(* CODESYS project tc3_harman_mesv2.6.10.library
   Author: Biro Csaba Attila
   Placeholder: Tc3_Harman_MES_Interface
   Title: Tc3_Harman_MES_Interface
   Version: 2.6.10
   Description: SAP-ME MES system interface library.
   Company: Harman

Project tree, tasks and I/O mapping:
  libraries: Tc2_Standard, * (Beckhoff Automation GmbH); Tc2_System, * (Beckhoff Automation GmbH); Tc2_TcpIp, * (Beckhoff Automation GmbH); Tc2_Utilities, * (Beckhoff Automation GmbH); Tc3_JsonXml, * (Beckhoff Automation GmbH); Tc3_Module, * (Beckhoff Automation GmbH); Tc3_Utilities_Extension, * (Harman)
  DUTs/
    data type E_TEST_STATE
    data type ENUM_MES_STATE
    data type ST_ASSEMBLY
    data type ST_ASSY_INFO
    data type ST_BOM
    data type ST_BOM_COMPONENT
    data type ST_GET_OP_STATE
    data type ST_INVENTORY
    data type ST_INVENTORY_LIST
    data type ST_MATERIAL
    data type ST_MATERIAL_INFO
    data type ST_MESDAT
    data type ST_MESDAT_ELEMENT
    data type ST_REQUEST
    data type ST_SET_ASSEMBLY
    data type ST_SHOPORDER
    data type ST_SHOPORDER_LIST
  FBs/
    function block FB_MES_INTERFACE_V2 [ST]: EXIT_SERVICE, GET_SERVICE_CONFIG, HIDE_SERVICE, LOCAL_INIT_SERVICE, REMOTE_INIT_SERVICE, SHOW_SERVICE, ASSY_ADD_MESDAT, ASSY_SAVE_MESDAT, ASSY_ADD_NCDAT, ASSY_SAVE_NCDAT, ASSEMBLE_BY_INVENTORY_LIST, CHECK_TIME_CONTROL, COMPLETE_SFC, GENERATE_SFC_BY_SO_AND_START, GET_CURRENT_OPERATION_STATE, GET_CUSTOM_DATA_BY_KEY, GET_INVENTORY_PARENT, GET_MAT_CUSTOM_DATA, GET_RECIPE_NAME_BY_OPERATION_JSON, GET_RECIPE_NAME_BY_OPERATION_XML, GET_SHOPORDER_BY_MAT, GET_TOTAL_BOM_BY_SO, IMPORT_AND_START_SFC, IMPORT_SFC, IS_VALID_INVENTORY_AND_IMPORT, MTERIAL_SETUP, SAVE_SFC_DATA, SCRAP_SFC, SIGNOFF_SFC, START_SFC, STOP_TIME_CONTROL, VALIDATE_IN_BOM, CREATE_XML_METH, GET_LOCAL_TIME, READ_XML_METH, FB_CALL_ACT
  FCs/
    function FC_GET_MATERIAL_FROM_HANDLE [ST]
    function FC_GET_REVISION_FROM_HANDLE [ST]
    function FC_REMOVE_HEADER [ST]
    function FC_REMOVE_STRING [ST]
  GVLs/
    global variables CONST_GVL
  TESTs/
    function GENERATE_MESDAT [ST]
    function GENERATE_NCDAT [ST]
    program HCP3_TEST_POU [ST]: FB_CALL_ACT
    program TEST_POU_1026_REPAIR [ST]: FB_CALL_ACT
    program TEST_POU_3026_SAVE_CF [ST]: FB_CALL_ACT
*)

// DUTs/E_TEST_STATE
TYPE E_TEST_STATE :
(
	PASSED:= 0,
	FAILED:= 1
):=FAILED;
END_TYPE

// DUTs/ENUM_MES_STATE
TYPE ENUM_MES_STATE :
(
	E_IDLE,
	E_CONNECTING,
	E_REQUEST_PROCESSING,
	E_REQUEST_PROCESSED,
	E_REQUEST_SEND,
	E_RESPONSE_RECIVED,
	E_RESPONSE_PROCESSING,
	E_RESPONSE_PROCESSED,
	E_DISCONNECTING,
	E_DONE,	
	E_ERROR		
):=E_IDLE;
END_TYPE

// DUTs/ST_ASSEMBLY
TYPE ST_ASSEMBLY :
STRUCT
	ASSEMBLY_READY		:STRING;
	ASSEMBLY_DONE		:STRING;
END_STRUCT
END_TYPE

// DUTs/ST_ASSY_INFO
TYPE ST_ASSY_INFO :
STRUCT
	ELEMENT:			ARRAY[1..9] OF ST_SET_ASSEMBLY;
END_STRUCT
END_TYPE

// DUTs/ST_BOM
TYPE ST_BOM :
STRUCT
	BOM_HANDLE:					STRING;
	BOMSTATUS:					STRING;
	DESCRIPTION:				STRING;
	SHOPORDER:					STRING;
	BOM_COMPONENTS:				ARRAY[0..19] OF ST_BOM_COMPONENT;
END_STRUCT
END_TYPE

// DUTs/ST_BOM_COMPONENT
TYPE ST_BOM_COMPONENT :
STRUCT
	BOM_COMPONENT_TYPE:				STRING;
	MATERIALS:						ARRAY[0..9] OF ST_MATERIAL;
	OPERATION:						STRING;
	QUANTITY:						STRING;
	SEQUENCE: 						STRING;
END_STRUCT
END_TYPE

// DUTs/ST_GET_OP_STATE
TYPE ST_GET_OP_STATE :
STRUCT
	ARCHIVE:		STRING;
	OP_INDEX:		STRING;
	OP_NAME:		STRING;
	SFC_STATE:		STRING;	
	OPEN_NC:		STRING;
	MAT_NO:			STRING;	
	REVISION:		STRING;
END_STRUCT
END_TYPE

// DUTs/ST_INVENTORY
TYPE ST_INVENTORY :
STRUCT
	DONE:			STRING;
	MAT_NO:			STRING;	
	REVISION:		STRING;
	SFC:			STRING;
	VALUES:			STRING;
END_STRUCT
END_TYPE

// DUTs/ST_INVENTORY_LIST
TYPE ST_INVENTORY_LIST :
STRUCT
	LIST:		ARRAY[0..9] OF ST_INVENTORY;
END_STRUCT
END_TYPE

// DUTs/ST_MATERIAL
TYPE ST_MATERIAL :
STRUCT
	MATERIAL:			STRING;
	REVISION:			STRING;
END_STRUCT
END_TYPE

// DUTs/ST_MATERIAL_INFO
TYPE ST_MATERIAL_INFO :
STRUCT
	MATNO:					STRING;
	REVISION:				STRING;
	SHOPORDER:				STRING;
	OPERATION:				STRING;
	RELEASECOUNT:			STRING;
END_STRUCT
END_TYPE

// DUTs/ST_MESDAT
TYPE ST_MESDAT :
STRUCT
	N:			INT;
	MESDAT:		ARRAY[1..200] OF ST_MESDAT_ELEMENT;
END_STRUCT
END_TYPE

// DUTs/ST_MESDAT_ELEMENT
TYPE ST_MESDAT_ELEMENT :
STRUCT
	RESPONSE_CODE:			STRING;		(* required in NC Data log - Error Id *)
	RESPONSE_DESCRIPTION:	STRING;		(* optional - Error description in NC Data log equal with DESCR *)
	CLIENT_DATE:			STRING;		(* required - Use the GET_LOCAL_TIME() method for generate in proper format. *)
	TEST_STATE:				STRING;		(* required - Use E_TEST_STATE value as string. *)
	TEST_STEP:				STRING;		(* required - Id of test step, (screw no, camera step...) *)
	DESCR:					STRING;		(* optional - Process step description, Error description in NC Data log *)
	UNIT:					STRING;		(* optional - Measurement unit *)
	VALUE:					STRING;		(* required - Measured data, if it Pass/Fail data only use 0 or 1 *)
	LL:						STRING;		(* optional - Lower limit *)
	UL:						STRING;		(* optional - Upper limit *)
END_STRUCT
END_TYPE

// DUTs/ST_REQUEST
TYPE ST_REQUEST :
STRUCT
	RESP_ACTION:		STRING;
	RESP_CODE:			STRING;
	ERR_MSG:			STRING[255];
END_STRUCT
END_TYPE

// DUTs/ST_SET_ASSEMBLY
TYPE ST_SET_ASSEMBLY :
STRUCT
	SFC:				STRING;
	MATNO:				STRING;
	REVISION:			STRING;
	INVENTORYID:		STRING;
	OPERATION:			STRING;
	RESOURCE:			STRING;
	DESCRIPTION:		STRING;
	BOM:				STRING;
	BOMREV:				STRING;
	SEQUENCE:			STRING;
	DATEASSEMBLED:		STRING;
	STRUCTUREPOSITION:	STRING;
	
	(*
	       <SET-ASSEMBLY>
            <SFC>614790420198010103089851</SFC>
            <MATNO>00003089851</MATNO>
            <REVISION>001</REVISION>
            <INVENTORYID>614790420198010103089851</INVENTORYID>
            <OPERATION>OP_ASSEMBLY_1</OPERATION>
            <RESOURCE>R_HUSZP5BRAFA11</RESOURCE>
            <DESCRIPTION>HOUSING HIGH RAM  B279 C1</DESCRIPTION>
            <BOM>00003561631_056</BOM>
            <BOMREV>001</BOMREV>
            <SEQUENCE>10</SEQUENCE>
            <DATEASSEMBLED>2/10/2020 10:59:04 PM</DATEASSEMBLED>
            <STRUCTUREPOSITION>0.0</STRUCTUREPOSITION>
          </SET-ASSEMBLY>
	*)
END_STRUCT
END_TYPE

// DUTs/ST_SHOPORDER
TYPE ST_SHOPORDER :
STRUCT
	HANDLE:				STRING;
	RELEASED:			STRING;
	STATUS:				STRING;
	QUANTITY:			STRING;
	SHOPORDER_TYPE:		STRING;
END_STRUCT
END_TYPE

// DUTs/ST_SHOPORDER_LIST
TYPE ST_SHOPORDER_LIST :
STRUCT
	LIST:		ARRAY[0..9] OF ST_SHOPORDER;
END_STRUCT
END_TYPE

// GVLs/CONST_GVL
VAR_GLOBAL CONSTANT
	DEFAULT_PRG_NAME:			STRING:='TwinCat3 - Build:v4024.17';
	DEFAULT_PRG_REV:			STRING:='v2.6.9';
END_VAR

// FBs/FB_MES_INTERFACE_V2
FUNCTION_BLOCK FB_MES_INTERFACE_V2
VAR_INPUT
	HOST:				T_IPV4ADDR := '';
	PORT:				UDINT;
	ENABLE:				BOOL;
	RESET:				BOOL;
	STX:				BYTE:= TCP_GVL.DEFAULT_STX;
	ETX:				BYTE:= TCP_GVL.DEFAULT_ETX;
	RESP:				REFERENCE TO ST_REQUEST;
	
	TEST_ADAPTER:		STRING;		//Adapter ID (Code)
	ADAPTER_ID:			STRING;		//Nest no. (1-5)
END_VAR
VAR_OUTPUT
	BUSY:				BOOL;
	READY:				BOOL;
	DONE:				BOOL;
	INTERFACE_CLOSED:	BOOL:=TRUE;
	ERROR:				BOOL;
	ERROR_ID:			UDINT;
END_VAR
VAR
	FB_TCP_IP_CLIENT:				FB_TCP_IP_CLIENT_LDAT;
	STATE:							ENUM_MES_STATE;
	
	INTERFACE_DIR:					STRING:='C:\Program Files\Harman\SAP-ME Interface';
	INTERFACE_FILE:					STRING:='SAP-ME Interface.exe';
	INTERFACE_ARG:					STRING:='initHMIAssy';
	
	EXECUTE:						BOOL;
	LOCAL_INIT:						BOOL;
	INIT:							BOOL;
	CB_MESSAGE:						UDINT;
	RT_EXECUTE, RT_RESET, RT_TCP_ERROR:R_TRIG;
	SYS_TIME_FB:					FB_LocalSystemTime;
	REQUEST_STRING:					STRING[DEFAULT_LDAT_LENGTH]:='';			
	RESPONSE_STRING:				STRING[DEFAULT_LDAT_LENGTH]:='';
	
	//================ XML =================
	FB_XML_PARSER: 			FB_XmlDomParser;
	OBJ_ROOT: 				SXmlNode;		
	
	// Base XML tags
	XML_HMIXML: 			SXmlNode;
	XML_PACKET: 			SXmlNode;	
	XML_BASICS: 			SXmlNode;		
	XML_ACTION: 			SXmlNode;
	XML_ARGUMENTS: 			SXmlNode;
	XML_RESULTS: 			SXmlNode;	
	XML_MSG: 				SXmlNode;	
	
	// Base response XML tags
	XML_RESCODE: 			SXmlNode;	
	XML_RESSTANDARDMESSAGE: SXmlNode;
	
	// Temporary container of RESTINFO for a later querys	
	XML_RESTINFO:			SXmlNode;
	
	// Request result inforamtion ErrorMessage, ResponseCode...
	XML_REQUEST_RESULT:		ST_REQUEST;	
	DEBUG:					STRING(10000);
	
	TP_RECONNECT:			TP;
	TON_INIT:				TON;
	FB_START_INTERFACE:		NT_StartProcess;
	eSubSystem: 			E_SubSystem:= E_SubSystem.LOGIC;
	FB_LOGGER:				FB_EventLogger:= (eSubsystem:= eSubsystem);
END_VAR

RT_EXECUTE(CLK:=EXECUTE);
RT_RESET(CLK:=RESET);
TP_RECONNECT(IN:=(FB_TCP_IP_CLIENT.CONNECTION_STATE<>ESOCKET_CONNECTED OR FB_TCP_IP_CLIENT.ERROR), PT:=T#250MS);
TON_INIT(IN:=INIT);	(* Delay for get configuration call *)
SYS_TIME_FB(bEnable:=TRUE,dwCycle:=1);

IF FB_TCP_IP_CLIENT.ERROR_ID<>0 THEN
	ERROR_ID:=FB_TCP_IP_CLIENT.ERROR_ID;
END_IF

BUSY:= STATE<>E_IDLE OR LOCAL_INIT OR INIT;
READY:= STATE=E_IDLE AND NOT INIT AND NOT INTERFACE_CLOSED;
ERROR:= STATE=E_ERROR;

IF RT_RESET.Q THEN
	//FB_LOGGER(sMsg:=CONCAT('Reseted externaly - ERROR_ID: ', UDINT_TO_STRING(ERROR_ID)), eSevr:=TcEventSeverity.Info);
	EXECUTE:=FALSE;
	ERROR_ID:= 0;
	STATE:=E_IDLE;
	REQUEST_STRING:= '';
	RESPONSE_STRING:= '';
	RESP.ERR_MSG:='';
	RESP.RESP_ACTION:='';
	RESP.RESP_CODE:='';
END_IF

(* Get MES configuration from interface *)
IF INIT THEN
	IF GET_SERVICE_CONFIG() THEN
		LOCAL_INIT:=FALSE;
		INIT:=FALSE;
	END_IF
END_IF

CASE STATE OF
	E_IDLE:
		IF RT_EXECUTE.Q THEN
			FB_TCP_IP_CLIENT.ENABLE:=TRUE;
			DONE:=FALSE;
			REQUEST_STRING:='';
			RESPONSE_STRING:='';
			CREATE_XML_METH();
			STATE:=E_CONNECTING;
		END_IF	
	E_CONNECTING:
		IF FB_TCP_IP_CLIENT.CONNECTION_STATE=ESOCKET_CONNECTED AND FB_TCP_IP_CLIENT.READY AND NOT FB_TCP_IP_CLIENT.BUSY THEN
			STATE:=E_REQUEST_PROCESSING;
		END_IF
		
	E_REQUEST_SEND:
		CB_MESSAGE:= FB_XML_PARSER.CopyDocument(REQUEST_STRING, SIZEOF(REQUEST_STRING));
		IF FB_TCP_IP_CLIENT.SEND(REQUEST_STRING, CB_MESSAGE, RESPONSE_STRING) THEN
			STATE:= E_RESPONSE_RECIVED;
		END_IF
		
	E_RESPONSE_RECIVED:
		READ_XML_METH();
		STATE:= E_RESPONSE_PROCESSING;
		MEMCPY(ADR(RESP),ADR(XML_REQUEST_RESULT), SIZEOF(XML_REQUEST_RESULT));
		
	E_DISCONNECTING:
		FB_TCP_IP_CLIENT.ENABLE:=FALSE;
		IF FB_TCP_IP_CLIENT.CONNECTION_STATE=ESOCKET_CONNECTED THEN
			STATE:=E_DONE;
		END_IF
	E_DONE:
		DONE:=TRUE;
		IF NOT EXECUTE THEN
			STATE:= E_IDLE;
		END_IF
		
	E_ERROR:
		//FB_LOGGER(sMsg:=CONCAT(CONCAT(CONCAT(CONCAT(CONCAT('Process done with issue. ERROR_ID: ', UDINT_TO_STRING(ERROR_ID)), ' Error message: '), XML_REQUEST_RESULT.ERR_MSG), ' Response code: '), XML_REQUEST_RESULT.RESP_CODE), eSevr:=TcEventSeverity.Error);
		EXECUTE:=FALSE;
		DONE:=FALSE;
		
END_CASE

IF ERROR_ID <> 0 THEN
	STATE:= E_ERROR;
END_IF

FB_CALL_ACT();

METHOD PUBLIC EXIT_SERVICE : BOOL
VAR
	XML_NODE:			SXmlNode;
END_VAR
CASE STATE OF
	E_IDLE:
		EXECUTE:=TRUE;
		
	E_REQUEST_PROCESSING:
		DEBUG:='';
		FB_XML_PARSER.AppendAttributeAsInt(XML_HMIXML,'operationIndex',0);
		FB_XML_PARSER.AppendAttributeAsInt(XML_HMIXML,'serviceId',2);		
		FB_XML_PARSER.SetChild(XML_ACTION,'1000001',FALSE);
		FB_XML_PARSER.CopyDocument(REQUEST_STRING, SIZEOF(REQUEST_STRING));
		STATE:= E_REQUEST_SEND;
		
	E_RESPONSE_PROCESSING:
		IF XML_REQUEST_RESULT.RESP_CODE = '0' THEN
			XML_RESTINFO:=FB_XML_PARSER.ChildByName(XML_RESULTS, 'RESTINFO');
			EXECUTE:=FALSE;
			STATE:= E_DISCONNECTING;
		ELSE
			MEMCPY(ADR(RESP),ADR(XML_REQUEST_RESULT), SIZEOF(XML_REQUEST_RESULT));
			ADSLOGSTR(ADSLOG_MSGTYPE_ERROR OR ADSLOG_MSGTYPE_LOG, 'SAP-ME error occured RESCODE: %s', CONCAT(CONCAT(RESP.RESP_CODE, ' ERR_MSG: '), RESP.ERR_MSG));
			EXECUTE:=FALSE;
			STATE:= E_DISCONNECTING;
		END_IF
	E_DONE: INTERFACE_CLOSED:=TRUE;
END_CASE
EXIT_SERVICE:= (STATE=E_DONE);
END_METHOD

METHOD PUBLIC GET_SERVICE_CONFIG : BOOL
VAR
	XML_NODE:			SXmlNode;
END_VAR
CASE STATE OF
	E_IDLE:
		EXECUTE:=TRUE;
		
	E_REQUEST_PROCESSING:
		DEBUG:='';
		FB_XML_PARSER.AppendAttributeAsInt(XML_HMIXML,'operationIndex',0);
		FB_XML_PARSER.AppendAttributeAsInt(XML_HMIXML,'serviceId',2);		
		FB_XML_PARSER.SetChild(XML_ACTION,'1000000',FALSE);
		FB_XML_PARSER.CopyDocument(REQUEST_STRING, SIZEOF(REQUEST_STRING));
		STATE:= E_REQUEST_SEND;
		
	E_RESPONSE_PROCESSING:
		IF XML_REQUEST_RESULT.RESP_CODE = '0' THEN
			XML_RESTINFO:=FB_XML_PARSER.ChildByName(XML_RESULTS, 'RESTINFO');
			EXECUTE:=FALSE;
			STATE:= E_DISCONNECTING;
		ELSE
			MEMCPY(ADR(RESP),ADR(XML_REQUEST_RESULT), SIZEOF(XML_REQUEST_RESULT));
			ADSLOGSTR(ADSLOG_MSGTYPE_ERROR OR ADSLOG_MSGTYPE_LOG, 'SAP-ME error occured RESCODE: %s', CONCAT(CONCAT(RESP.RESP_CODE, ' ERR_MSG: '), RESP.ERR_MSG));
			EXECUTE:=FALSE;
			STATE:= E_DISCONNECTING;
		END_IF
END_CASE
GET_SERVICE_CONFIG:= (STATE=E_DONE);
END_METHOD

METHOD PUBLIC HIDE_SERVICE : BOOL
VAR
	XML_NODE:			SXmlNode;
END_VAR
CASE STATE OF
	E_IDLE:
		EXECUTE:=TRUE;
		
	E_REQUEST_PROCESSING:
		DEBUG:='';
		FB_XML_PARSER.AppendAttributeAsInt(XML_HMIXML,'operationIndex',0);
		FB_XML_PARSER.AppendAttributeAsInt(XML_HMIXML,'serviceId',2);		
		FB_XML_PARSER.SetChild(XML_ACTION,'1000003',FALSE);
		FB_XML_PARSER.CopyDocument(REQUEST_STRING, SIZEOF(REQUEST_STRING));
		STATE:= E_REQUEST_SEND;
		
	E_RESPONSE_PROCESSING:
		IF XML_REQUEST_RESULT.RESP_CODE = '0' THEN
			XML_RESTINFO:=FB_XML_PARSER.ChildByName(XML_RESULTS, 'RESTINFO');
			EXECUTE:=FALSE;
			STATE:= E_DISCONNECTING;
		ELSE
			MEMCPY(ADR(RESP),ADR(XML_REQUEST_RESULT), SIZEOF(XML_REQUEST_RESULT));
			ADSLOGSTR(ADSLOG_MSGTYPE_ERROR OR ADSLOG_MSGTYPE_LOG, 'SAP-ME error occured RESCODE: %s', CONCAT(CONCAT(RESP.RESP_CODE, ' ERR_MSG: '), RESP.ERR_MSG));
			EXECUTE:=FALSE;
			STATE:= E_DISCONNECTING;
		END_IF
	E_DONE: INTERFACE_CLOSED:=TRUE;
END_CASE
HIDE_SERVICE:= (STATE=E_DONE);
END_METHOD

METHOD PUBLIC LOCAL_INIT_SERVICE : BOOL
LOCAL_INIT:=TRUE;
TON_INIT.PT:=T#3S;
INIT:=TRUE;
INTERFACE_CLOSED:=FALSE;
LOCAL_INIT_SERVICE:= STATE=E_DONE;
END_METHOD

METHOD PUBLIC REMOTE_INIT_SERVICE : BOOL
INIT:=TRUE;
TON_INIT.PT:=T#0S;
INTERFACE_CLOSED:=FALSE;
REMOTE_INIT_SERVICE:= STATE=E_DONE;
END_METHOD

METHOD PUBLIC SHOW_SERVICE : BOOL
VAR
	XML_NODE:			SXmlNode;
END_VAR
CASE STATE OF
	E_IDLE:
		EXECUTE:=TRUE;
		
	E_REQUEST_PROCESSING:
		DEBUG:='';
		FB_XML_PARSER.AppendAttributeAsInt(XML_HMIXML,'operationIndex',0);
		FB_XML_PARSER.AppendAttributeAsInt(XML_HMIXML,'serviceId',2);		
		FB_XML_PARSER.SetChild(XML_ACTION,'1000002',FALSE);
		FB_XML_PARSER.CopyDocument(REQUEST_STRING, SIZEOF(REQUEST_STRING));
		STATE:= E_REQUEST_SEND;
		
	E_RESPONSE_PROCESSING:
		IF XML_REQUEST_RESULT.RESP_CODE = '0' THEN
			XML_RESTINFO:=FB_XML_PARSER.ChildByName(XML_RESULTS, 'RESTINFO');
			EXECUTE:=FALSE;
			STATE:= E_DISCONNECTING;
		ELSE
			MEMCPY(ADR(RESP),ADR(XML_REQUEST_RESULT), SIZEOF(XML_REQUEST_RESULT));
			ADSLOGSTR(ADSLOG_MSGTYPE_ERROR OR ADSLOG_MSGTYPE_LOG, 'SAP-ME error occured RESCODE: %s', CONCAT(CONCAT(RESP.RESP_CODE, ' ERR_MSG: '), RESP.ERR_MSG));
			EXECUTE:=FALSE;
			STATE:= E_DISCONNECTING;
		END_IF
	E_DONE: INTERFACE_CLOSED:=TRUE;
END_CASE
SHOW_SERVICE:= (STATE=E_DONE);
END_METHOD

METHOD PUBLIC ASSY_ADD_MESDAT : BOOL
VAR_INPUT
	DATA:				REFERENCE TO ST_MESDAT_ELEMENT;
END_VAR
VAR
	XML_SET:			SXmlNode;
	XML_CLIENTDATE:		SXmlNode;
	XML_TESTSTATE:		SXmlNode;
	XML_TESTSTEP:		SXmlNode;	
	XML_DESCR:			SXmlNode;
	XML_TESTVALUE:		SXmlNode;		
	XML_UNIT:			SXmlNode;	
	XML_LOWERLIMIT:		SXmlNode;	
	XML_UPPERLIMIT:		SXmlNode;	
END_VAR
ASSY_ADD_MESDAT:=FALSE;
XML_SET := FB_XML_PARSER.AppendNode(XML_ARGUMENTS, 'SET');	
		
XML_CLIENTDATE := FB_XML_PARSER.AppendNode(XML_SET, 'CLIENTDATE'); //Req
XML_TESTSTATE := FB_XML_PARSER.AppendNode(XML_SET, 'TESTSTATE');//Req
XML_TESTSTEP := FB_XML_PARSER.AppendNode(XML_SET, 'TESTSTEP');//Req
XML_DESCR := FB_XML_PARSER.AppendNode(XML_SET, 'DESCR'); //Optional
XML_TESTVALUE := FB_XML_PARSER.AppendNode(XML_SET, 'TESTVALUE');//Req
XML_UNIT := FB_XML_PARSER.AppendNode(XML_SET, 'UNIT');	//Optional
XML_LOWERLIMIT := FB_XML_PARSER.AppendNode(XML_SET, 'LOWERLIMIT'); //Optional
XML_UPPERLIMIT := FB_XML_PARSER.AppendNode(XML_SET, 'UPPERLIMIT'); //Optional

FB_XML_PARSER.SetChild(XML_CLIENTDATE, DATA.CLIENT_DATE, FALSE);
FB_XML_PARSER.SetChild(XML_TESTSTATE,DATA.TEST_STATE, FALSE);			
FB_XML_PARSER.SetChild(XML_TESTSTEP, DATA.TEST_STEP, FALSE);					
FB_XML_PARSER.SetChild(XML_DESCR, DATA.DESCR, FALSE);				
FB_XML_PARSER.SetChild(XML_TESTVALUE, DATA.VALUE, FALSE);					
FB_XML_PARSER.SetChild(XML_UNIT, DATA.UNIT, FALSE);							
FB_XML_PARSER.SetChild(XML_LOWERLIMIT, DATA.LL, FALSE);							
FB_XML_PARSER.SetChild(XML_UPPERLIMIT, DATA.UL, FALSE);

ASSY_ADD_MESDAT:=TRUE;
END_METHOD

METHOD PUBLIC ASSY_SAVE_MESDAT : BOOL
VAR_INPUT
	SFC:					STRING;					//Product Serial Number
	INDEX:					INT;					//Operation index
	DATA:					REFERENCE TO ST_MESDAT;	//Measurement data.	
END_VAR
VAR_OUTPUT
	
END_VAR
VAR
	XML_NODE:				SXmlNode;
	XML_TESTADAPTER:		SXmlNode;
	XML_ADAPTERID:			SXmlNode;
	XML_PROGRAMNAME: 		SXmlNode;	
	XML_PROGREV:			SXmlNode;
			
	CNT:					INT:=1;
END_VAR
CASE STATE OF
	E_IDLE:
		IF DATA.N>=1 AND DATA.N<=200 THEN
			EXECUTE:=TRUE;
		ELSE
			// TODO: If data array is empty return and log error message.
			ASSY_SAVE_MESDAT:=TRUE;
		END_IF
		
	E_REQUEST_PROCESSING:		
		FB_XML_PARSER.AppendAttributeAsInt(XML_HMIXML,'operationIndex',INDEX);
		FB_XML_PARSER.AppendAttributeAsInt(XML_HMIXML,'serviceId',2);	
			
		XML_NODE:= FB_XML_PARSER.AppendNode(XML_ARGUMENTS, 'SFC');
		XML_TESTADAPTER:= FB_XML_PARSER.AppendNode(XML_ARGUMENTS, 'TESTADAPTER'); //Req
		XML_ADAPTERID:= FB_XML_PARSER.AppendNode(XML_ARGUMENTS, 'FIXTUREID'); //Req
		XML_PROGRAMNAME:= FB_XML_PARSER.AppendNode(XML_ARGUMENTS, 'PROGRAMID'); //Optional
		XML_PROGREV:= FB_XML_PARSER.AppendNode(XML_ARGUMENTS, 'PROGRAMREV'); //Optional
		
		FB_XML_PARSER.SetChild(XML_ACTION,'3523', FALSE);
		
		FB_XML_PARSER.SetChild(XML_NODE, SFC, FALSE);
		FB_XML_PARSER.SetChild(XML_TESTADAPTER, TEST_ADAPTER, FALSE);
		FB_XML_PARSER.SetChild(XML_ADAPTERID, ADAPTER_ID, FALSE);
		FB_XML_PARSER.SetChild(XML_PROGRAMNAME, DEFAULT_PRG_NAME, FALSE);	
		FB_XML_PARSER.SetChild(XML_PROGREV, DEFAULT_PRG_REV, FALSE);	
		
		FOR CNT:=1 TO (DATA.N) DO
			ASSY_ADD_MESDAT(DATA.MESDAT[CNT]);			
		END_FOR
		
		STATE:= E_REQUEST_SEND;
		
	E_RESPONSE_PROCESSING:
		IF XML_REQUEST_RESULT.RESP_CODE = '0' THEN		
			EXECUTE:=FALSE;
			STATE:= E_DISCONNECTING;
		ELSE
			MEMCPY(ADR(RESP),ADR(XML_REQUEST_RESULT), SIZEOF(XML_REQUEST_RESULT));
			ADSLOGSTR(ADSLOG_MSGTYPE_ERROR OR ADSLOG_MSGTYPE_LOG, 'SAP-ME error occured RESCODE: %s', CONCAT(CONCAT(RESP.RESP_CODE, ' ERR_MSG: '), RESP.ERR_MSG));
			EXECUTE:=FALSE;
			STATE:= E_DISCONNECTING;
		END_IF

END_CASE
ASSY_SAVE_MESDAT:= (STATE=E_DONE);
END_METHOD

METHOD PUBLIC ASSY_ADD_NCDAT : BOOL
VAR_INPUT
	DATA:				REFERENCE TO ST_MESDAT_ELEMENT;
END_VAR
VAR
	XML_SET:			SXmlNode;
	XML_TESTSTATE:		SXmlNode;
	XML_TESTSTEP:		SXmlNode;	
	XML_RESPCODE:		SXmlNode;
	XML_RESPDESC:		SXmlNode;	
	XML_DESCR:			SXmlNode;
	XML_TESTVALUE:		SXmlNode;
	XML_LOWERLIMIT:		SXmlNode;	
	XML_UPPERLIMIT:		SXmlNode;	
END_VAR
ASSY_ADD_NCDAT:=FALSE;
XML_SET := FB_XML_PARSER.AppendNode(XML_ARGUMENTS, 'SET');	
		
XML_TESTSTATE := FB_XML_PARSER.AppendNode(XML_SET, 'TESTSTATE');
XML_TESTSTEP := FB_XML_PARSER.AppendNode(XML_SET, 'TESTSTEP');
XML_RESPCODE := FB_XML_PARSER.AppendNode(XML_SET, 'RESPONSECODE');
XML_RESPDESC := FB_XML_PARSER.AppendNode(XML_SET, 'RESPONSECODEDESCR');
XML_DESCR := FB_XML_PARSER.AppendNode(XML_SET, 'DESCR');
XML_TESTVALUE := FB_XML_PARSER.AppendNode(XML_SET, 'TESTVALUE');
XML_LOWERLIMIT := FB_XML_PARSER.AppendNode(XML_SET, 'LOWERLIMIT');
XML_UPPERLIMIT := FB_XML_PARSER.AppendNode(XML_SET, 'UPPERLIMIT');

FB_XML_PARSER.SetChild(XML_TESTSTATE, DATA.TEST_STATE, FALSE);			
FB_XML_PARSER.SetChild(XML_TESTSTEP, DATA.TEST_STEP, FALSE);
FB_XML_PARSER.SetChild(XML_RESPCODE, DATA.RESPONSE_CODE, FALSE);			
FB_XML_PARSER.SetChild(XML_RESPDESC, DATA.RESPONSE_DESCRIPTION, FALSE);					
FB_XML_PARSER.SetChild(XML_DESCR, DATA.DESCR, FALSE);				
FB_XML_PARSER.SetChild(XML_TESTVALUE, DATA.VALUE, FALSE);					
FB_XML_PARSER.SetChild(XML_LOWERLIMIT, DATA.LL, FALSE);							
FB_XML_PARSER.SetChild(XML_UPPERLIMIT, DATA.UL, FALSE);	

ASSY_ADD_NCDAT:=TRUE;
END_METHOD

METHOD PUBLIC ASSY_SAVE_NCDAT : BOOL
VAR_INPUT
	SFC:					STRING;					//Product Serial Number
	INDEX:					INT;					//Operation index
	DATA:					REFERENCE TO ST_MESDAT;	//Measurement data.	
END_VAR
VAR_OUTPUT
	
END_VAR
VAR
	XML_SFC:				SXmlNode;
	XML_TESTADAPTER:		SXmlNode;
	XML_ADAPTERID:			SXmlNode;
	XML_CLIENTDATE:			SXmlNode;
	CLIENT_DATE:			STRING;	
	CNT:					INT:=1;
END_VAR
CLIENT_DATE:= GET_LOCAL_TIME();
CASE STATE OF
	E_IDLE:
		IF DATA.N>=1 AND DATA.N<=200 THEN
			EXECUTE:=TRUE;
		ELSE
			// TODO: If data array is empty generate unknown error... just for fail safe NC Logging
			DATA.N:=1;
			DATA.MESDAT[1].CLIENT_DATE:=GET_LOCAL_TIME();
			DATA.MESDAT[1].DESCR:='Unknown TwinCAT error - No data found in NC-Data container.';
			DATA.MESDAT[1].LL:='0';
			DATA.MESDAT[1].RESPONSE_CODE:='16003';
			DATA.MESDAT[1].RESPONSE_DESCRIPTION:='Unknown TwinCAT error - No data found in NC-Data container.';
			DATA.MESDAT[1].TEST_STATE:='1';
			DATA.MESDAT[1].TEST_STEP:='-1';
			DATA.MESDAT[1].UL:='0';
			DATA.MESDAT[1].UNIT:='Dig';
			DATA.MESDAT[1].VALUE:='-1';
			
			EXECUTE:=TRUE;
		END_IF
		
	E_REQUEST_PROCESSING:		
		CLIENT_DATE:=GET_LOCAL_TIME();
		FB_XML_PARSER.AppendAttributeAsInt(XML_HMIXML,'operationIndex',INDEX);
		FB_XML_PARSER.AppendAttributeAsInt(XML_HMIXML,'serviceId',2);	
			
		XML_SFC:= FB_XML_PARSER.AppendNode(XML_ARGUMENTS, 'SFC');
		XML_CLIENTDATE := FB_XML_PARSER.AppendNode(XML_ARGUMENTS, 'CLIENTDATE');
		XML_TESTADAPTER:= FB_XML_PARSER.AppendNode(XML_ARGUMENTS, 'TESTADAPTER');
		XML_ADAPTERID:= FB_XML_PARSER.AppendNode(XML_ARGUMENTS, 'FIXTUREID');
		
		FB_XML_PARSER.SetChild(XML_ACTION,'3503', FALSE);
		
		FB_XML_PARSER.SetChild(XML_SFC, SFC, FALSE);
		FB_XML_PARSER.SetChild(XML_CLIENTDATE, CLIENT_DATE, FALSE);
		FB_XML_PARSER.SetChild(XML_TESTADAPTER, TEST_ADAPTER, FALSE);
		FB_XML_PARSER.SetChild(XML_ADAPTERID, ADAPTER_ID, FALSE);	
		
		FOR CNT:=1 TO (DATA.N) DO
			ASSY_ADD_NCDAT(DATA.MESDAT[CNT]);			
		END_FOR
		
		STATE:= E_REQUEST_SEND;
		
	E_RESPONSE_PROCESSING:
		IF XML_REQUEST_RESULT.RESP_CODE = '0' THEN		
			EXECUTE:=FALSE;
			STATE:= E_DISCONNECTING;
		ELSE
			MEMCPY(ADR(RESP),ADR(XML_REQUEST_RESULT), SIZEOF(XML_REQUEST_RESULT));
			ADSLOGSTR(ADSLOG_MSGTYPE_ERROR OR ADSLOG_MSGTYPE_LOG, 'SAP-ME error occured RESCODE: %s', CONCAT(CONCAT(RESP.RESP_CODE, ' ERR_MSG: '), RESP.ERR_MSG));
			EXECUTE:=FALSE;
			STATE:= E_DISCONNECTING;
		END_IF

END_CASE
ASSY_SAVE_NCDAT:= (STATE=E_DONE);
END_METHOD

METHOD PUBLIC ASSEMBLE_BY_INVENTORY_LIST : BOOL
VAR_INPUT
	SFC:				STRING;
	INDEX:				INT;
	INVENTORY_LIST:		ST_INVENTORY_LIST;
END_VAR
VAR
	XML_NODE:			SXmlNode;
	XML_SET:			SXmlNode;
	XML_INVENTORY_ID:	SXmlNode;
	XML_INVENTORI_MAT:	SXmlNode;
	XML_INVENTORI_REV:	SXmlNode;
	
	CNT:				INT;
END_VAR
CASE STATE OF
	E_IDLE:
		EXECUTE:=TRUE;
		
	E_REQUEST_PROCESSING:
		DEBUG:='';
		FB_XML_PARSER.AppendAttributeAsInt(XML_HMIXML,'operationIndex',INDEX);
		FB_XML_PARSER.AppendAttributeAsInt(XML_HMIXML,'serviceId',2);		
		FB_XML_PARSER.SetChild(XML_ACTION,'2138',FALSE);
		XML_NODE := FB_XML_PARSER.AppendNode(XML_ARGUMENTS, 'SFC');
		FB_XML_PARSER.SetChild(XML_NODE,SFC,FALSE);
		FOR CNT:=0 TO 9 BY 1 DO
			IF INVENTORY_LIST.LIST[CNT].SFC<>'' AND LEN(INVENTORY_LIST.LIST[CNT].MAT_NO)=11 AND LEN(INVENTORY_LIST.LIST[CNT].REVISION)=3 THEN
				XML_SET := FB_XML_PARSER.AppendNode(XML_ARGUMENTS, 'SET');
					XML_INVENTORY_ID := FB_XML_PARSER.AppendNode(XML_SET, 'INVENTORYID');
					FB_XML_PARSER.SetChild(XML_INVENTORY_ID,INVENTORY_LIST.LIST[CNT].SFC,FALSE);
					XML_INVENTORI_MAT := FB_XML_PARSER.AppendNode(XML_SET, 'MATNO');
					FB_XML_PARSER.SetChild(XML_INVENTORI_MAT,INVENTORY_LIST.LIST[CNT].MAT_NO,FALSE);
					XML_INVENTORI_REV := FB_XML_PARSER.AppendNode(XML_SET, 'MATNO_REV');
					FB_XML_PARSER.SetChild(XML_INVENTORI_REV,INVENTORY_LIST.LIST[CNT].REVISION,FALSE);
			END_IF			
		END_FOR;
		
		FB_XML_PARSER.CopyDocument(REQUEST_STRING, SIZEOF(REQUEST_STRING));
		DEBUG:=REQUEST_STRING;
		STATE:= E_REQUEST_SEND;
		
	E_RESPONSE_PROCESSING:
		IF XML_REQUEST_RESULT.RESP_CODE = '0' THEN
			XML_RESTINFO:=FB_XML_PARSER.ChildByName(XML_RESULTS, 'RESTINFO');		
			EXECUTE:=FALSE;
			STATE:= E_DISCONNECTING;
		ELSE
			MEMCPY(ADR(RESP),ADR(XML_REQUEST_RESULT), SIZEOF(XML_REQUEST_RESULT));
			ADSLOGSTR(ADSLOG_MSGTYPE_ERROR OR ADSLOG_MSGTYPE_LOG, 'SAP-ME error occured RESCODE: %s', CONCAT(CONCAT(RESP.RESP_CODE, ' ERR_MSG: '), RESP.ERR_MSG));
			EXECUTE:=FALSE;
			STATE:= E_DISCONNECTING;
		END_IF

END_CASE
ASSEMBLE_BY_INVENTORY_LIST:= (STATE=E_DONE);
END_METHOD

METHOD PUBLIC CHECK_TIME_CONTROL : BOOL
VAR_INPUT
	SFC:				STRING;
	CONTROLTYPE:		STRING; //required Time Control Type Filter
	RESULT:				REFERENCE TO BOOL; //result is set to high if the sfc have active time control
	INDEX:				INT;
END_VAR
VAR
	XML_NODE:			SXmlNode;
END_VAR
CASE STATE OF
	E_IDLE:
		EXECUTE:=TRUE;
		
	E_REQUEST_PROCESSING:
		DEBUG:='';
		FB_XML_PARSER.AppendAttributeAsInt(XML_HMIXML,'operationIndex',INDEX);
		FB_XML_PARSER.AppendAttributeAsInt(XML_HMIXML,'serviceId',2);		
		FB_XML_PARSER.SetChild(XML_ACTION,'2034',FALSE);
		(* Set arguments *)
		XML_NODE := FB_XML_PARSER.AppendNode(XML_ARGUMENTS, 'SFC');
		FB_XML_PARSER.SetChild(XML_NODE,SFC,FALSE);
		XML_NODE := FB_XML_PARSER.AppendNode(XML_ARGUMENTS, 'CONTROLTYPE');
		FB_XML_PARSER.SetChild(XML_NODE,CONTROLTYPE,FALSE);
		
		FB_XML_PARSER.CopyDocument(REQUEST_STRING, SIZEOF(REQUEST_STRING));
		DEBUG:=REQUEST_STRING;
		STATE:= E_REQUEST_SEND;
		
	E_RESPONSE_PROCESSING:
		IF XML_REQUEST_RESULT.RESP_CODE = '0' THEN
			RESULT:=TRUE;
			XML_RESTINFO:=FB_XML_PARSER.ChildByName(XML_RESULTS, 'RESTINFO');
			EXECUTE:=FALSE;
			STATE:= E_DISCONNECTING;
		ELSE
			MEMCPY(ADR(RESP),ADR(XML_REQUEST_RESULT), SIZEOF(XML_REQUEST_RESULT));
			RESULT:=FALSE;
			ADSLOGSTR(ADSLOG_MSGTYPE_ERROR OR ADSLOG_MSGTYPE_LOG, 'SAP-ME error occured RESCODE: %s', CONCAT(CONCAT(RESP.RESP_CODE, ' ERR_MSG: '), RESP.ERR_MSG));
			EXECUTE:=FALSE;
			STATE:= E_DISCONNECTING;
		END_IF

END_CASE
CHECK_TIME_CONTROL:= (STATE=E_DONE);
END_METHOD

METHOD PUBLIC COMPLETE_SFC : BOOL
VAR_INPUT
	SFC:				STRING;				//Product Serial Number	
	INDEX:				INT;
	TEST_STATE:			E_TEST_STATE;		//0:PASSED,1:FAILED
END_VAR
VAR
	XML_SFC:				SXmlNode;
	XML_TESTSTATE:			SXmlNode;
	XML_TESTADAPTER:		SXmlNode;
	XML_ADAPTERID:			SXmlNode;
	XML_CLIENTDATE:			SXmlNode;	
	XML_PROGRAMNAME:		SXmlNode;	
	STRING_TEST_STATE:		STRING;	
	CLIENT_DATE_STRING:		STRING;
END_VAR
CASE STATE OF
	E_IDLE:
		EXECUTE:=TRUE;
		
	E_REQUEST_PROCESSING:
		CLIENT_DATE_STRING:=GET_LOCAL_TIME();
		STRING_TEST_STATE:=INT_TO_STRING(TEST_STATE);
		
		FB_XML_PARSER.AppendAttributeAsInt(XML_HMIXML,'operationIndex',INDEX);
		FB_XML_PARSER.AppendAttributeAsInt(XML_HMIXML,'serviceId',2);
		FB_XML_PARSER.SetChild(XML_ACTION,'3011', FALSE);
		
		XML_SFC:= FB_XML_PARSER.AppendNode(XML_ARGUMENTS, 'SFC');		
		XML_TESTSTATE:= FB_XML_PARSER.AppendNode(XML_ARGUMENTS, 'TESTSTATE');
		XML_TESTADAPTER:= FB_XML_PARSER.AppendNode(XML_ARGUMENTS, 'TESTADAPTER');
		XML_ADAPTERID:= FB_XML_PARSER.AppendNode(XML_ARGUMENTS, 'ADAPTERID');
		XML_CLIENTDATE:= FB_XML_PARSER.AppendNode(XML_ARGUMENTS, 'CLIENTDATE');
		XML_PROGRAMNAME:= FB_XML_PARSER.AppendNode(XML_ARGUMENTS, 'PROGRAMNAME');
		
		
		FB_XML_PARSER.SetChild(XML_SFC, SFC, FALSE);
		FB_XML_PARSER.SetChild(XML_TESTSTATE, STRING_TEST_STATE, FALSE);
		FB_XML_PARSER.SetChild(XML_TESTADAPTER, TEST_ADAPTER, FALSE);
		FB_XML_PARSER.SetChild(XML_ADAPTERID, ADAPTER_ID, FALSE);
		FB_XML_PARSER.SetChild(XML_CLIENTDATE, CLIENT_DATE_STRING, FALSE);
		FB_XML_PARSER.SetChild(XML_PROGRAMNAME, DEFAULT_PRG_NAME, FALSE);
		
		STATE:= E_REQUEST_SEND;
		
	E_RESPONSE_PROCESSING:
		IF XML_REQUEST_RESULT.RESP_CODE = '0' THEN
			XML_RESTINFO:=FB_XML_PARSER.ChildByName(XML_RESULTS, 'RESTINFO');		
			EXECUTE:=FALSE;
			STATE:= E_DISCONNECTING;
		ELSE
			MEMCPY(ADR(RESP),ADR(XML_REQUEST_RESULT), SIZEOF(XML_REQUEST_RESULT));
			ADSLOGSTR(ADSLOG_MSGTYPE_ERROR OR ADSLOG_MSGTYPE_LOG, 'SAP-ME error occured RESCODE: %s', CONCAT(CONCAT(RESP.RESP_CODE, ' ERR_MSG: '), RESP.ERR_MSG));
			EXECUTE:=FALSE;
			STATE:= E_DISCONNECTING;
		END_IF

END_CASE
COMPLETE_SFC:= (STATE=E_DONE);
END_METHOD

METHOD PUBLIC GENERATE_SFC_BY_SO_AND_START : BOOL
VAR_INPUT
	MATERIAL:				ST_MATERIAL_INFO;
	INSEQUENCE:				STRING;
	AUTOCOMPLETE:			STRING;
	LEADING_SFC:			REFERENCE TO STRING;
	INDEX:					INT;
END_VAR
VAR
	XML_MATNO:				SXmlNode;
	XML_REVISION:			SXmlNode;
	XML_SHOPORDER:			SXmlNode;
	XML_INSEQUENCE:			SXmlNode;
	XML_AUTOCOMPLETE:		SXmlNode;	
	XML_RESPONSE_NODE: 		SXmlNode;
END_VAR
CASE STATE OF
	E_IDLE:
		EXECUTE:=TRUE;
		
	E_REQUEST_PROCESSING:
		DEBUG:='';
		FB_XML_PARSER.AppendAttributeAsInt(XML_HMIXML,'operationIndex',INDEX);
		FB_XML_PARSER.AppendAttributeAsInt(XML_HMIXML,'serviceId',2);		
		FB_XML_PARSER.SetChild(XML_ACTION,'1004',FALSE);
		
		XML_MATNO := FB_XML_PARSER.AppendNode(XML_ARGUMENTS, 'MATNO');
		XML_REVISION := FB_XML_PARSER.AppendNode(XML_ARGUMENTS, 'MATNO_REV');
		XML_SHOPORDER := FB_XML_PARSER.AppendNode(XML_ARGUMENTS, 'SHOPORDER');
		XML_INSEQUENCE := FB_XML_PARSER.AppendNode(XML_ARGUMENTS, 'INSEQUENCE');
		XML_AUTOCOMPLETE := FB_XML_PARSER.AppendNode(XML_ARGUMENTS, 'AUTOCOMPLETE');
		
		FB_XML_PARSER.SetChild(XML_MATNO, MATERIAL.MATNO, FALSE);
		FB_XML_PARSER.SetChild(XML_REVISION, MATERIAL.REVISION, FALSE);
		FB_XML_PARSER.SetChild(XML_SHOPORDER, MATERIAL.SHOPORDER, FALSE);
		FB_XML_PARSER.SetChild(XML_INSEQUENCE, INSEQUENCE, FALSE);
		FB_XML_PARSER.SetChild(XML_AUTOCOMPLETE, AUTOCOMPLETE, FALSE);
		
		FB_XML_PARSER.CopyDocument(REQUEST_STRING, SIZEOF(REQUEST_STRING));
		DEBUG:=REQUEST_STRING;
		STATE:= E_REQUEST_SEND;
		
	E_RESPONSE_PROCESSING:
		IF XML_REQUEST_RESULT.RESP_CODE = '0' THEN
			XML_RESTINFO:=FB_XML_PARSER.ChildByName(XML_RESULTS, 'RESTINFO');
			XML_RESPONSE_NODE:=FB_XML_PARSER.ChildByName(XML_RESULTS, 'SFC');	
			LEADING_SFC:= FB_XML_PARSER.NodeText(XML_RESPONSE_NODE);		
			EXECUTE:=FALSE;
			STATE:= E_DISCONNECTING;
		ELSE
			MEMCPY(ADR(RESP),ADR(XML_REQUEST_RESULT), SIZEOF(XML_REQUEST_RESULT));
			ADSLOGSTR(ADSLOG_MSGTYPE_ERROR OR ADSLOG_MSGTYPE_LOG, 'SAP-ME error occured RESCODE: %s', CONCAT(CONCAT(RESP.RESP_CODE, ' ERR_MSG: '), RESP.ERR_MSG));
			EXECUTE:=FALSE;
			STATE:= E_DISCONNECTING;
		END_IF

END_CASE
GENERATE_SFC_BY_SO_AND_START:= (STATE=E_DONE);
END_METHOD

METHOD PUBLIC GET_CURRENT_OPERATION_STATE : BOOL
VAR_INPUT
	SFC:				STRING;
	INDEX:				INT;
	RESULT:				REFERENCE TO ST_GET_OP_STATE;
END_VAR
VAR
	XML_NODE:				SXmlNode;
END_VAR
CASE STATE OF
	E_IDLE:
		EXECUTE:=TRUE;
		
	E_REQUEST_PROCESSING:
		FB_XML_PARSER.AppendAttributeAsInt(XML_HMIXML,'operationIndex',INDEX);
		FB_XML_PARSER.AppendAttributeAsInt(XML_HMIXML,'serviceId',2);			
		FB_XML_PARSER.SetChild(XML_ACTION,'1026',FALSE);
		
		XML_NODE := FB_XML_PARSER.AppendNode(XML_ARGUMENTS, 'SFC');
		FB_XML_PARSER.SetChild(XML_NODE,SFC,FALSE);
		
		FB_XML_PARSER.CopyDocument(REQUEST_STRING, SIZEOF(REQUEST_STRING));
		STATE:= E_REQUEST_SEND;
		
	E_RESPONSE_PROCESSING:
		IF XML_REQUEST_RESULT.RESP_CODE = '0' OR XML_REQUEST_RESULT.RESP_CODE = '377' THEN
			XML_NODE:=FB_XML_PARSER.ChildByName(XML_RESULTS, 'MATNO');
			FB_XML_PARSER.CopyNodeText(XML_NODE, RESULT.MAT_NO, SIZEOF(RESULT.MAT_NO));
			XML_NODE:=FB_XML_PARSER.ChildByName(XML_RESULTS, 'MATNO_REV');
			FB_XML_PARSER.CopyNodeText(XML_NODE, RESULT.REVISION, SIZEOF(RESULT.REVISION));
			XML_NODE:=FB_XML_PARSER.ChildByName(XML_RESULTS, 'OPENNC');
			FB_XML_PARSER.CopyNodeText(XML_NODE, RESULT.OPEN_NC, SIZEOF(RESULT.OPEN_NC));
			XML_NODE:=FB_XML_PARSER.ChildByName(XML_RESULTS, 'OPERATION_INDEX');
			FB_XML_PARSER.CopyNodeText(XML_NODE, RESULT.OP_INDEX, SIZEOF(RESULT.OP_INDEX));
			XML_NODE:=FB_XML_PARSER.ChildByName(XML_RESULTS, 'OPERATION');
			FB_XML_PARSER.CopyNodeText(XML_NODE, RESULT.OP_NAME, SIZEOF(RESULT.OP_NAME));
			XML_NODE:=FB_XML_PARSER.ChildByName(XML_RESULTS, 'SFC_STATE');
			FB_XML_PARSER.CopyNodeText(XML_NODE, RESULT.SFC_STATE, SIZEOF(RESULT.SFC_STATE));	
			XML_NODE:=FB_XML_PARSER.ChildByName(XML_RESULTS, 'ARCHIVE');
			FB_XML_PARSER.CopyNodeText(XML_NODE, RESULT.ARCHIVE, SIZEOF(RESULT.ARCHIVE));
			
			EXECUTE:=FALSE;
			STATE:= E_DISCONNECTING;
		ELSE
			MEMCPY(ADR(RESP),ADR(XML_REQUEST_RESULT), SIZEOF(XML_REQUEST_RESULT));
			ADSLOGSTR(ADSLOG_MSGTYPE_ERROR OR ADSLOG_MSGTYPE_LOG, 'SAP-ME error occured RESCODE: %s', CONCAT(CONCAT(RESP.RESP_CODE, ' ERR_MSG: '), RESP.ERR_MSG));
			EXECUTE:=FALSE;
			STATE:= E_DISCONNECTING;
		END_IF

END_CASE
GET_CURRENT_OPERATION_STATE:= (STATE=E_DONE);
END_METHOD

METHOD PUBLIC GET_CUSTOM_DATA_BY_KEY : BOOL
VAR_INPUT
	KEY:					STRING;
	RESULT:					REFERENCE TO STRING(1000);
END_VAR
VAR_OUTPUT
	
END_VAR
VAR
	XML_NODE:				SXmlNode;
END_VAR
XML_NODE:= FB_XML_PARSER.ChildByName(XML_RESTINFO, KEY);
RESULT:= FB_XML_PARSER.NodeText(XML_NODE);
GET_CUSTOM_DATA_BY_KEY:=TRUE;
RETURN;
END_METHOD

METHOD PUBLIC GET_INVENTORY_PARENT : BOOL
VAR_INPUT
	SFC:				STRING;
	INDEX:				INT;
	RESULT:				REFERENCE TO STRING;	
END_VAR
VAR
	XML_NODE:			SXmlNode;
	XML_SFC:			SXmlNode;
END_VAR
CASE STATE OF
	E_IDLE:
		EXECUTE:=TRUE;
		
	E_REQUEST_PROCESSING:
		FB_XML_PARSER.AppendAttributeAsInt(XML_HMIXML,'operationIndex',INDEX);
		FB_XML_PARSER.AppendAttributeAsInt(XML_HMIXML,'serviceId',2);		
		FB_XML_PARSER.SetChild(XML_ACTION,'3005',FALSE);
		
		XML_NODE := FB_XML_PARSER.AppendNode(XML_ARGUMENTS, 'INVENTORYID');
		FB_XML_PARSER.SetChild(XML_NODE,SFC,FALSE);
		
		FB_XML_PARSER.CopyDocument(REQUEST_STRING, SIZEOF(REQUEST_STRING));
		STATE:= E_REQUEST_SEND;
		
	E_RESPONSE_PROCESSING:
		IF XML_REQUEST_RESULT.RESP_CODE = '0' OR XML_REQUEST_RESULT.RESP_CODE = '587' OR XML_REQUEST_RESULT.RESP_CODE = '597' THEN
			XML_SFC:=FB_XML_PARSER.ChildByName(XML_RESULTS, 'PARENTSFC');
			FB_XML_PARSER.CopyNodeText(XML_SFC, RESULT, SIZEOF(RESULT));	
			
			EXECUTE:=FALSE;
			STATE:= E_DISCONNECTING;
		ELSE
			MEMCPY(ADR(RESP),ADR(XML_REQUEST_RESULT), SIZEOF(XML_REQUEST_RESULT));
			ADSLOGSTR(ADSLOG_MSGTYPE_ERROR OR ADSLOG_MSGTYPE_LOG, 'SAP-ME error occured RESCODE: %s', CONCAT(CONCAT(RESP.RESP_CODE, ' ERR_MSG: '), RESP.ERR_MSG));
			EXECUTE:=FALSE;
			STATE:= E_DISCONNECTING;
		END_IF

END_CASE
GET_INVENTORY_PARENT:= (STATE=E_DONE);
END_METHOD

METHOD PUBLIC GET_MAT_CUSTOM_DATA : BOOL
VAR_INPUT
	MATERIAL:			REFERENCE TO ST_MATERIAL;
	INDEX:				INT;
END_VAR
VAR
	XML_NODE:			SXmlNode;
END_VAR
CASE STATE OF
	E_IDLE:
		EXECUTE:=TRUE;
		
	E_REQUEST_PROCESSING:
		DEBUG:='';
		FB_XML_PARSER.AppendAttributeAsInt(XML_HMIXML,'operationIndex',INDEX);
		FB_XML_PARSER.AppendAttributeAsInt(XML_HMIXML,'serviceId',2);		
		FB_XML_PARSER.SetChild(XML_ACTION,'1037',FALSE);
		XML_NODE := FB_XML_PARSER.AppendNode(XML_ARGUMENTS, 'MATNO');
		FB_XML_PARSER.SetChild(XML_NODE, MATERIAL.MATERIAL,FALSE);
		XML_NODE := FB_XML_PARSER.AppendNode(XML_ARGUMENTS, 'MATNO_REV');
		FB_XML_PARSER.SetChild(XML_NODE, MATERIAL.REVISION,FALSE);
		
		FB_XML_PARSER.CopyDocument(REQUEST_STRING, SIZEOF(REQUEST_STRING));
		DEBUG:=REQUEST_STRING;
		STATE:= E_REQUEST_SEND;
		
	E_RESPONSE_PROCESSING:
		IF XML_REQUEST_RESULT.RESP_CODE = '0' THEN
			XML_RESTINFO:=XML_RESULTS;
			EXECUTE:=FALSE;
			STATE:= E_DISCONNECTING;
		ELSE
			MEMCPY(ADR(RESP),ADR(XML_REQUEST_RESULT), SIZEOF(XML_REQUEST_RESULT));
			ADSLOGSTR(ADSLOG_MSGTYPE_ERROR OR ADSLOG_MSGTYPE_LOG, 'SAP-ME error occured RESCODE: %s', CONCAT(CONCAT(RESP.RESP_CODE, ' ERR_MSG: '), RESP.ERR_MSG));
			EXECUTE:=FALSE;
			STATE:= E_DISCONNECTING;
		END_IF

END_CASE
GET_MAT_CUSTOM_DATA:= (STATE=E_DONE);
END_METHOD

METHOD PUBLIC GET_RECIPE_NAME_BY_OPERATION_JSON : BOOL
VAR_INPUT
	KEY:					STRING;
	RESULT:					REFERENCE TO STRING;
END_VAR
VAR
	XML_NODE:				SXmlNode;
	JSON_TEXT:				STRING(512);
	JSON_PARSER:			FB_JsonDomParser;
	JSON_DOC:				SJsonValue;
	JSON_PROP: 				SJsonValue;
	JSON_HAS_MEMBER: 		BOOL;
END_VAR
XML_NODE:= FB_XML_PARSER.ChildByName(XML_RESTINFO, 'RECIPE_DATA');
JSON_TEXT:=FB_XML_PARSER.NodeText(XML_NODE);

//Repleace ' to "
WHILE FIND(JSON_TEXT,'$'')>0 DO JSON_TEXT:=REPLACE(JSON_TEXT, '$"', 1, FIND(JSON_TEXT,'$'')); END_WHILE

JSON_DOC := JSON_PARSER.ParseDocument(JSON_TEXT);
JSON_HAS_MEMBER := JSON_PARSER.HasMember(JSON_DOC, KEY);
IF JSON_HAS_MEMBER THEN
	JSON_HAS_MEMBER:= FALSE;
	JSON_PROP:= JSON_PARSER.FindMember(JSON_DOC, KEY);
	RESULT:= JSON_PARSER.GetString(JSON_PROP);
ELSE
	MEMSET(ADR(RESULT), 0, SIZEOF(RESULT));	
END_IF
GET_RECIPE_NAME_BY_OPERATION_JSON:=TRUE;
END_METHOD

METHOD PUBLIC GET_RECIPE_NAME_BY_OPERATION_XML : BOOL
VAR_INPUT
	KEY:					STRING;
	RESULT:					REFERENCE TO STRING;
END_VAR
VAR
	XML_NODE:				SXmlNode;
	XML_OP_RECIPE:			SXmlNode;
END_VAR
XML_NODE:= FB_XML_PARSER.ChildByName(XML_RESTINFO, 'RECIPE_DATA');
XML_OP_RECIPE:= FB_XML_PARSER.ChildByName(XML_NODE, KEY);
RESULT:= FB_XML_PARSER.NodeText(XML_OP_RECIPE);	
GET_RECIPE_NAME_BY_OPERATION_XML:=TRUE;
END_METHOD

METHOD PUBLIC GET_SHOPORDER_BY_MAT : BOOL
VAR_INPUT
	MATERIAL:				REFERENCE TO ST_MATERIAL;
	RELEASE:				STRING;
	INDEX:					INT;
	RESULT:					REFERENCE TO ST_SHOPORDER_LIST;
END_VAR
VAR
	XML_NODE:				SXmlNode;
	XML_SHOPORDER_INFO:		SXmlNode;
	XML_ITERATOR:			SXmlIterator;
	
	CNT:					INT:=0;
END_VAR
CASE STATE OF
	E_IDLE:
		EXECUTE:=TRUE;
		
	E_REQUEST_PROCESSING:
		FB_XML_PARSER.AppendAttributeAsInt(XML_HMIXML,'operationIndex',INDEX);
		FB_XML_PARSER.AppendAttributeAsInt(XML_HMIXML,'serviceId',2);		
		FB_XML_PARSER.SetChild(XML_ACTION,'3009',FALSE);
		
		XML_NODE := FB_XML_PARSER.AppendNode(XML_ARGUMENTS, 'MATNO');
		FB_XML_PARSER.SetChild(XML_NODE,MATERIAL.MATERIAL,FALSE);
		XML_NODE := FB_XML_PARSER.AppendNode(XML_ARGUMENTS, 'MATNO_REV');
		FB_XML_PARSER.SetChild(XML_NODE,MATERIAL.REVISION,FALSE);
		XML_NODE := FB_XML_PARSER.AppendNode(XML_ARGUMENTS, 'RELEASECOUNT');
		FB_XML_PARSER.SetChild(XML_NODE,RELEASE,FALSE);
		
		FB_XML_PARSER.CopyDocument(REQUEST_STRING, SIZEOF(REQUEST_STRING));
		STATE:= E_REQUEST_SEND;
		
	E_RESPONSE_PROCESSING:
		IF XML_REQUEST_RESULT.RESP_CODE = '0' THEN
			XML_RESTINFO:=FB_XML_PARSER.ChildByName(XML_RESULTS, 'RESTINFO');
			XML_ITERATOR:=FB_XML_PARSER.BeginByName(XML_RESULTS,'SET');
			(* Iterate all tag in result and get BOM data from each element *)
			WHILE NOT FB_XML_PARSER.IsEnd(XML_ITERATOR) DO
				XML_NODE:=FB_XML_PARSER.Node(XML_ITERATOR);
				IF CNT>9 THEN
					(* Escape if more than 10 shoporder is in the list... *)
					EXECUTE:=FALSE;
					STATE:= E_DISCONNECTING;
				ELSE
					(* Decapsulate shoporder data from selected tag... *)
						//TODO: Need string function to get the proper shoporder string
					XML_SHOPORDER_INFO:= FB_XML_PARSER.ChildByName(XML_NODE, 'SHOPORDERHANDLE');
					RESULT.LIST[CNT].HANDLE:= FC_REMOVE_HEADER(FB_XML_PARSER.NodeText(XML_SHOPORDER_INFO));		
			  
				  	XML_SHOPORDER_INFO:= FB_XML_PARSER.ChildByName(XML_NODE, 'SHOPORDERTOBUILD');
				  	RESULT.LIST[CNT].QUANTITY:= FB_XML_PARSER.NodeText(XML_SHOPORDER_INFO);
				  	XML_SHOPORDER_INFO:= FB_XML_PARSER.ChildByName(XML_NODE, 'SHOPORDERRELEASED');
				  	RESULT.LIST[CNT].RELEASED:= FB_XML_PARSER.NodeText(XML_SHOPORDER_INFO);						 
				  	XML_SHOPORDER_INFO:= FB_XML_PARSER.ChildByName(XML_NODE, 'SHOPORDERSTATUS');
				  	RESULT.LIST[CNT].STATUS:= FB_XML_PARSER.NodeText(XML_SHOPORDER_INFO);						  
				  	XML_SHOPORDER_INFO:= FB_XML_PARSER.ChildByName(XML_NODE, 'SHOPORDERTYPE');
				  	RESULT.LIST[CNT].SHOPORDER_TYPE:= FB_XML_PARSER.NodeText(XML_SHOPORDER_INFO);		
				  
			  		CNT:=CNT+1;
					XML_ITERATOR:= FB_XML_PARSER.NextByName(XML_ITERATOR, 'SET');
				END_IF
			END_WHILE
			
			EXECUTE:=FALSE;
			STATE:= E_DISCONNECTING;
		ELSE
			MEMCPY(ADR(RESP),ADR(XML_REQUEST_RESULT), SIZEOF(XML_REQUEST_RESULT));
			ADSLOGSTR(ADSLOG_MSGTYPE_ERROR OR ADSLOG_MSGTYPE_LOG, 'SAP-ME error occured RESCODE: %s', CONCAT(CONCAT(RESP.RESP_CODE, ' ERR_MSG: '), RESP.ERR_MSG));
			EXECUTE:=FALSE;
			STATE:= E_DISCONNECTING;
		END_IF

END_CASE
GET_SHOPORDER_BY_MAT:= (STATE=E_DONE);
END_METHOD

METHOD PUBLIC GET_TOTAL_BOM_BY_SO : BOOL
VAR_INPUT
	SHOPORDER:				STRING;
	INDEX:					INT;
	RESULT:					REFERENCE TO ST_BOM;
END_VAR
VAR
	XML_NODE:				SXmlNode;
	XML_BOM_COMPONENT_INFO:	SXmlNode;
	XML_ITERATOR:			SXmlIterator;
	
	CNT:					INT:=0;
	TAG_NAME:				STRING;
	CNT_ALT:				INT:=1;
END_VAR
CASE STATE OF
	E_IDLE:
		EXECUTE:=TRUE;
		
	E_REQUEST_PROCESSING:
		FB_XML_PARSER.AppendAttributeAsInt(XML_HMIXML,'operationIndex',INDEX);
		FB_XML_PARSER.AppendAttributeAsInt(XML_HMIXML,'serviceId',2);		
		FB_XML_PARSER.SetChild(XML_ACTION,'3008',FALSE);
		
		XML_NODE := FB_XML_PARSER.AppendNode(XML_ARGUMENTS, 'SHOPORDER');
		FB_XML_PARSER.SetChild(XML_NODE,SHOPORDER,FALSE);
		
		FB_XML_PARSER.CopyDocument(REQUEST_STRING, SIZEOF(REQUEST_STRING));
		STATE:= E_REQUEST_SEND;
		
	E_RESPONSE_PROCESSING:
		IF XML_REQUEST_RESULT.RESP_CODE = '0' THEN
			XML_RESTINFO:=FB_XML_PARSER.ChildByName(XML_RESULTS, 'RESTINFO');
			
			(* Get default BOM data *)
			XML_NODE:= FB_XML_PARSER.ChildByName(XML_RESULTS, 'BOMHANDLE');
			RESULT.BOM_HANDLE:=FB_XML_PARSER.NodeText(XML_NODE);
			XML_NODE:=FB_XML_PARSER.ChildByName(XML_RESULTS, 'BOMSTATUS');
			RESULT.BOMSTATUS:=FB_XML_PARSER.NodeText(XML_NODE);
			XML_NODE:=FB_XML_PARSER.ChildByName(XML_RESULTS, 'DESCRIPTION');
			RESULT.DESCRIPTION:=FB_XML_PARSER.NodeText(XML_NODE);
			XML_NODE:=FB_XML_PARSER.ChildByName(XML_RESULTS, 'SHOPORDER');
			RESULT.SHOPORDER:=FB_XML_PARSER.NodeText(XML_NODE);
			
			XML_ITERATOR:=FB_XML_PARSER.BeginByName(XML_RESULTS,'SET');
			(* Iterate all tag in result and get BOM data from each element *)
			WHILE NOT FB_XML_PARSER.IsEnd(XML_ITERATOR) DO
				XML_NODE:=FB_XML_PARSER.Node(XML_ITERATOR);
				IF CNT>19 THEN
					(* Escape if more than 10 shoporder is in the list... *)
					EXECUTE:=FALSE;
					STATE:= E_DISCONNECTING;
				ELSE
					(* Decapsulate shoporder data from selected tag... *)
					XML_BOM_COMPONENT_INFO:= FB_XML_PARSER.ChildByName(XML_NODE, 'BOMCOMPONENTTYPE');
					RESULT.BOM_COMPONENTS[CNT].BOM_COMPONENT_TYPE:= FB_XML_PARSER.NodeText(XML_BOM_COMPONENT_INFO);		
			  
				  	XML_BOM_COMPONENT_INFO:= FB_XML_PARSER.ChildByName(XML_NODE, 'QUANTITY');
				  	RESULT.BOM_COMPONENTS[CNT].QUANTITY:= FB_XML_PARSER.NodeText(XML_BOM_COMPONENT_INFO);
			  
				  	XML_BOM_COMPONENT_INFO:= FB_XML_PARSER.ChildByName(XML_NODE, 'OPERATION');
				  	RESULT.BOM_COMPONENTS[CNT].OPERATION:= FB_XML_PARSER.NodeText(XML_BOM_COMPONENT_INFO);			
			 
				  	XML_BOM_COMPONENT_INFO:= FB_XML_PARSER.ChildByName(XML_NODE, 'SEQUENCE');
				  	RESULT.BOM_COMPONENTS[CNT].SEQUENCE:= FB_XML_PARSER.NodeText(XML_BOM_COMPONENT_INFO);		
				  
				  	//Bom compnents...
				  	XML_BOM_COMPONENT_INFO:= FB_XML_PARSER.ChildByName(XML_NODE, 'MATERIALHANDLE');

				  	RESULT.BOM_COMPONENTS[CNT].MATERIALS[0].MATERIAL:= FC_GET_MATERIAL_FROM_HANDLE(FC_REMOVE_HEADER(FB_XML_PARSER.NodeText(XML_BOM_COMPONENT_INFO)));		
				  	RESULT.BOM_COMPONENTS[CNT].MATERIALS[0].REVISION:= FC_GET_REVISION_FROM_HANDLE(FC_REMOVE_HEADER(FB_XML_PARSER.NodeText(XML_BOM_COMPONENT_INFO)));	
					
					CNT_ALT:=1;
					FOR CNT_ALT:=1 TO 9 BY 1 DO
						TAG_NAME:= CONCAT('ALTERMATERIALHANDLE_',INT_TO_STRING(CNT_ALT-1));
						XML_BOM_COMPONENT_INFO:= FB_XML_PARSER.ChildByName(XML_NODE,TAG_NAME);
						RESULT.BOM_COMPONENTS[CNT].MATERIALS[CNT_ALT].MATERIAL:= FC_GET_MATERIAL_FROM_HANDLE(FC_REMOVE_HEADER(FB_XML_PARSER.NodeText(XML_BOM_COMPONENT_INFO)));		
						RESULT.BOM_COMPONENTS[CNT].MATERIALS[CNT_ALT].REVISION:= FC_GET_REVISION_FROM_HANDLE(FC_REMOVE_HEADER(FB_XML_PARSER.NodeText(XML_BOM_COMPONENT_INFO)));
					END_FOR;
					
			  		CNT:=CNT+1;
					XML_ITERATOR:= FB_XML_PARSER.NextByName(XML_ITERATOR, 'SET');
				END_IF
			END_WHILE
			
			EXECUTE:=FALSE;
			STATE:= E_DISCONNECTING;
		ELSE
			MEMCPY(ADR(RESP),ADR(XML_REQUEST_RESULT), SIZEOF(XML_REQUEST_RESULT));
			ADSLOGSTR(ADSLOG_MSGTYPE_ERROR OR ADSLOG_MSGTYPE_LOG, 'SAP-ME error occured RESCODE: %s', CONCAT(CONCAT(RESP.RESP_CODE, ' ERR_MSG: '), RESP.ERR_MSG));
			EXECUTE:=FALSE;
			STATE:= E_DISCONNECTING;
		END_IF

END_CASE
GET_TOTAL_BOM_BY_SO:= (STATE=E_DONE);
END_METHOD

METHOD PUBLIC IMPORT_AND_START_SFC : BOOL
VAR_INPUT
	SFC:				STRING;
	INDEX:				INT;
END_VAR
VAR
	XML_NODE:				SXmlNode;
END_VAR
CASE STATE OF
	E_IDLE:
		EXECUTE:=TRUE;
		
	E_REQUEST_PROCESSING:
		FB_XML_PARSER.AppendAttributeAsInt(XML_HMIXML,'operationIndex',INDEX);
		FB_XML_PARSER.AppendAttributeAsInt(XML_HMIXML,'serviceId',2);			
		FB_XML_PARSER.SetChild(XML_ACTION,'28',FALSE);
		XML_NODE := FB_XML_PARSER.AppendNode(XML_ARGUMENTS, 'SFC');
		FB_XML_PARSER.SetChild(XML_NODE,SFC,FALSE);
		
		FB_XML_PARSER.CopyDocument(REQUEST_STRING, SIZEOF(REQUEST_STRING));
		STATE:= E_REQUEST_SEND;
		
	E_RESPONSE_PROCESSING:
		IF XML_REQUEST_RESULT.RESP_CODE = '0' THEN
			XML_RESTINFO:=FB_XML_PARSER.ChildByName(XML_RESULTS, 'RESTINFO');		
			EXECUTE:=FALSE;
			STATE:= E_DISCONNECTING;
		ELSE
			MEMCPY(ADR(RESP),ADR(XML_REQUEST_RESULT), SIZEOF(XML_REQUEST_RESULT));
			ADSLOGSTR(ADSLOG_MSGTYPE_ERROR OR ADSLOG_MSGTYPE_LOG, 'SAP-ME error occured RESCODE: %s', CONCAT(CONCAT(RESP.RESP_CODE, ' ERR_MSG: '), RESP.ERR_MSG));
			EXECUTE:=FALSE;
			STATE:= E_DISCONNECTING;
		END_IF

END_CASE
IMPORT_AND_START_SFC:= (STATE=E_DONE);
END_METHOD

METHOD PUBLIC IMPORT_SFC : BOOL
VAR_INPUT
	SFC:				STRING;
	INDEX:				INT;
	RESULT:				REFERENCE TO ST_INVENTORY;
END_VAR
VAR
	XML_NODE:			SXmlNode;
	XML_SFC_INFO:		SXmlNode;
END_VAR
CASE STATE OF
	E_IDLE:
		EXECUTE:=TRUE;
		
	E_REQUEST_PROCESSING:
		DEBUG:='';
		FB_XML_PARSER.AppendAttributeAsInt(XML_HMIXML,'operationIndex',INDEX);
		FB_XML_PARSER.AppendAttributeAsInt(XML_HMIXML,'serviceId',2);		
		FB_XML_PARSER.SetChild(XML_ACTION,'28',FALSE);
		XML_NODE := FB_XML_PARSER.AppendNode(XML_ARGUMENTS, 'SFC');
		FB_XML_PARSER.SetChild(XML_NODE,SFC,FALSE);
		
		FB_XML_PARSER.CopyDocument(REQUEST_STRING, SIZEOF(REQUEST_STRING));
		DEBUG:=REQUEST_STRING;
		STATE:= E_REQUEST_SEND;
		
	E_RESPONSE_PROCESSING:
		IF XML_REQUEST_RESULT.RESP_CODE = '0' THEN
			XML_RESTINFO:=FB_XML_PARSER.ChildByName(XML_RESULTS, 'RESTINFO');
			XML_NODE:=FB_XML_PARSER.ChildByName(XML_RESULTS, 'SET');
			
			XML_SFC_INFO:= FB_XML_PARSER.ChildByName(XML_NODE, 'MATNO');
			RESULT.MAT_NO:= FC_REMOVE_HEADER(FB_XML_PARSER.NodeText(XML_SFC_INFO));
			XML_SFC_INFO:= FB_XML_PARSER.ChildByName(XML_NODE, 'MATNO_REV');
			RESULT.REVISION:= FB_XML_PARSER.NodeText(XML_SFC_INFO);
			XML_SFC_INFO:= FB_XML_PARSER.ChildByName(XML_NODE, 'SFC');
			RESULT.SFC:= FB_XML_PARSER.NodeText(XML_SFC_INFO);						 
			XML_SFC_INFO:= FB_XML_PARSER.ChildByName(XML_NODE, 'VALUES');
			RESULT.VALUES:= FB_XML_PARSER.NodeText(XML_SFC_INFO);
				RESULT.DONE:= 'FALSE';
			EXECUTE:=FALSE;
			STATE:= E_DISCONNECTING;
		ELSE
			MEMCPY(ADR(RESP),ADR(XML_REQUEST_RESULT), SIZEOF(XML_REQUEST_RESULT));
			ADSLOGSTR(ADSLOG_MSGTYPE_ERROR OR ADSLOG_MSGTYPE_LOG, 'SAP-ME error occured RESCODE: %s', CONCAT(CONCAT(RESP.RESP_CODE, ' ERR_MSG: '), RESP.ERR_MSG));
			EXECUTE:=FALSE;
			STATE:= E_DISCONNECTING;
		END_IF
END_CASE
IMPORT_SFC:= (STATE=E_DONE);
END_METHOD

METHOD PUBLIC IS_VALID_INVENTORY_AND_IMPORT : BOOL
VAR_INPUT
	INVENTORYID:		STRING;
	INDEX:				INT;
	RESULT:				REFERENCE TO ST_INVENTORY;
END_VAR
VAR
	XML_SET:				SXmlNode;
	XML_DONE:				SXmlNode;
	XML_MATNO:				SXmlNode;
	XML_MATNO_REV:			SXmlNode;
	XML_SFC:				SXmlNode;
	XML_VALUES:				SXmlNode;	
	
	XML_NODE:				SXmlNode;
END_VAR
CASE STATE OF
	E_IDLE:
		EXECUTE:=TRUE;
		
	E_REQUEST_PROCESSING:
		FB_XML_PARSER.AppendAttributeAsInt(XML_HMIXML,'operationIndex',INDEX);
		FB_XML_PARSER.AppendAttributeAsInt(XML_HMIXML,'serviceId',2);			
		FB_XML_PARSER.SetChild(XML_ACTION,'2011',FALSE);
		
		XML_NODE := FB_XML_PARSER.AppendNode(XML_ARGUMENTS, 'INVENTORYID');
		FB_XML_PARSER.SetChild(XML_NODE,INVENTORYID,FALSE);
		
		FB_XML_PARSER.CopyDocument(REQUEST_STRING, SIZEOF(REQUEST_STRING));
		STATE:= E_REQUEST_SEND;
		
	E_RESPONSE_PROCESSING:
		IF XML_REQUEST_RESULT.RESP_CODE = '0' THEN		
			XML_SET:=FB_XML_PARSER.ChildByName(XML_RESULTS, 'SET');
		
			XML_DONE:=FB_XML_PARSER.ChildByName(XML_SET, 'DONE');
			XML_MATNO:=FB_XML_PARSER.ChildByName(XML_SET, 'MATNO');
			XML_MATNO_REV:=FB_XML_PARSER.ChildByName(XML_SET, 'MATNO_REV');
			XML_SFC:=FB_XML_PARSER.ChildByName(XML_SET, 'SFC');
			XML_VALUES:=FB_XML_PARSER.ChildByName(XML_SET, 'VALUES');
		
			FB_XML_PARSER.CopyNodeText(XML_DONE, RESULT.DONE, SIZEOF(RESULT.DONE));
			FB_XML_PARSER.CopyNodeText(XML_MATNO, RESULT.MAT_NO, SIZEOF(RESULT.MAT_NO));
			FB_XML_PARSER.CopyNodeText(XML_MATNO_REV, RESULT.REVISION, SIZEOF(RESULT.REVISION));	
			FB_XML_PARSER.CopyNodeText(XML_SFC, RESULT.SFC, SIZEOF(RESULT.SFC));
			FB_XML_PARSER.CopyNodeText(XML_VALUES, RESULT.VALUES, SIZEOF(RESULT.VALUES));
	
			EXECUTE:=FALSE;
			STATE:= E_DISCONNECTING;
		ELSE
			MEMCPY(ADR(RESP),ADR(XML_REQUEST_RESULT), SIZEOF(XML_REQUEST_RESULT));
			ADSLOGSTR(ADSLOG_MSGTYPE_ERROR OR ADSLOG_MSGTYPE_LOG, 'SAP-ME error occured RESCODE: %s', CONCAT(CONCAT(RESP.RESP_CODE, ' ERR_MSG: '), RESP.ERR_MSG));
			EXECUTE:=FALSE;
			STATE:= E_DISCONNECTING;
		END_IF

END_CASE
IS_VALID_INVENTORY_AND_IMPORT:= (STATE=E_DONE);
END_METHOD

METHOD PUBLIC MTERIAL_SETUP : BOOL
VAR_INPUT
	MATERIAL:				REFERENCE TO ST_MATERIAL;
	RELEASE:				STRING;
	INDEX:					INT;
END_VAR
VAR
	XML_NODE:				SXmlNode;
END_VAR
CASE STATE OF
	E_IDLE:
		EXECUTE:=TRUE;
		
	E_REQUEST_PROCESSING:
		FB_XML_PARSER.AppendAttributeAsInt(XML_HMIXML,'operationIndex',INDEX);
		FB_XML_PARSER.AppendAttributeAsInt(XML_HMIXML,'serviceId',2);		
		FB_XML_PARSER.SetChild(XML_ACTION,'3009',FALSE);
		
		XML_NODE := FB_XML_PARSER.AppendNode(XML_ARGUMENTS, 'MATNO');
		FB_XML_PARSER.SetChild(XML_NODE,MATERIAL.MATERIAL,FALSE);
		XML_NODE := FB_XML_PARSER.AppendNode(XML_ARGUMENTS, 'MATNO_REV');
		FB_XML_PARSER.SetChild(XML_NODE,MATERIAL.REVISION,FALSE);
		XML_NODE := FB_XML_PARSER.AppendNode(XML_ARGUMENTS, 'RELEASECOUNT');
		FB_XML_PARSER.SetChild(XML_NODE,RELEASE,FALSE);
		
		FB_XML_PARSER.CopyDocument(REQUEST_STRING, SIZEOF(REQUEST_STRING));
		STATE:= E_REQUEST_SEND;
		
	E_RESPONSE_PROCESSING:
		IF XML_REQUEST_RESULT.RESP_CODE = '0' THEN
			XML_RESTINFO:=FB_XML_PARSER.ChildByName(XML_RESULTS, 'RESTINFO');
			EXECUTE:=FALSE;
			STATE:= E_DISCONNECTING;
		ELSE
			MEMCPY(ADR(RESP),ADR(XML_REQUEST_RESULT), SIZEOF(XML_REQUEST_RESULT));
			ADSLOGSTR(ADSLOG_MSGTYPE_ERROR OR ADSLOG_MSGTYPE_LOG, 'SAP-ME error occured RESCODE: %s', CONCAT(CONCAT(RESP.RESP_CODE, ' ERR_MSG: '), RESP.ERR_MSG));
			EXECUTE:=FALSE;
			STATE:= E_DISCONNECTING;
		END_IF

END_CASE
MTERIAL_SETUP:= (STATE=E_DONE);
END_METHOD

METHOD PUBLIC SAVE_SFC_DATA : BOOL
VAR_INPUT
	SFC:					STRING; // barcode
	ADAPTERID:				STRING;	// adapter id
	INDEX:					INT;	// operation index
	SFCATTRIBUTE:			STRING; // custom field name
	ATTRIBUTEVALUE:			STRING; // custom field value
END_VAR
VAR
	XML_NODE:				SXmlNode;//XML structure
	XML_SET_NODE:			SXmlNode;// XML SET
	XML_SFC_NODE:			SXmlNode;// XML SFC NODE
	XML_ADAPTERID_NODE:		SXmlNode;// XML ADAPTERID NODE
	XML_SFCATTRIBUTE_NODE:	SXmlNode;// XML SFCATTRIBUTE NODE
	XML_ATTRIBUTEVALUE_NODE:SXmlNode;// XML ATTRIBUTEVALUE NODE
END_VAR
CASE STATE OF
	E_IDLE:
		EXECUTE:=TRUE;
		
	E_REQUEST_PROCESSING:
		FB_XML_PARSER.AppendAttributeAsInt(XML_HMIXML,'operationIndex',INDEX);
		FB_XML_PARSER.AppendAttributeAsInt(XML_HMIXML,'serviceId',2);			
		FB_XML_PARSER.SetChild(XML_ACTION,'3026',FALSE);
		
		XML_SFC_NODE := FB_XML_PARSER.AppendNode(XML_ARGUMENTS, 'SFC');
		FB_XML_PARSER.SetChild(XML_SFC_NODE,SFC,FALSE);
		
		XML_NODE := FB_XML_PARSER.AppendNode(XML_ARGUMENTS, 'ADAPTERID');
		FB_XML_PARSER.SetChild(XML_NODE,ADAPTERID,FALSE);
		
		XML_SET_NODE := FB_XML_PARSER.AppendNode(XML_ARGUMENTS, 'SET');
		
		XML_SFCATTRIBUTE_NODE := FB_XML_PARSER.AppendNode(XML_SET_NODE, 'SFCATTRIBUTE');
		XML_ATTRIBUTEVALUE_NODE := FB_XML_PARSER.AppendNode(XML_SET_NODE, 'ATTRIBUTEVALUE');
		
		FB_XML_PARSER.SetChild(XML_SFCATTRIBUTE_NODE,SFCATTRIBUTE,FALSE);
		FB_XML_PARSER.SetChild(XML_ATTRIBUTEVALUE_NODE,ATTRIBUTEVALUE,FALSE);
		
		FB_XML_PARSER.CopyDocument(REQUEST_STRING, SIZEOF(REQUEST_STRING));
		STATE:= E_REQUEST_SEND;
		
	E_RESPONSE_PROCESSING:
		IF XML_REQUEST_RESULT.RESP_CODE = '0' THEN
			XML_RESTINFO:=FB_XML_PARSER.ChildByName(XML_RESULTS, 'ARGUMENTS');
			EXECUTE:=FALSE;
			STATE:= E_DISCONNECTING;
		ELSE
			MEMCPY(ADR(RESP),ADR(XML_REQUEST_RESULT), SIZEOF(XML_REQUEST_RESULT));
			ADSLOGSTR(ADSLOG_MSGTYPE_ERROR OR ADSLOG_MSGTYPE_LOG, 'SAP-ME error occured RESCODE: %s', CONCAT(CONCAT(RESP.RESP_CODE, ' ERR_MSG: '), RESP.ERR_MSG));
			EXECUTE:=FALSE;
			STATE:= E_DISCONNECTING;
		END_IF
END_CASE
SAVE_SFC_DATA:=(STATE=E_DONE);
END_METHOD

METHOD PUBLIC SCRAP_SFC : BOOL
VAR_INPUT
	SFC:				STRING;
	INDEX:				INT;			
END_VAR
VAR
	XML_NODE:			SXmlNode;
END_VAR
CASE STATE OF
	E_IDLE:
		EXECUTE:=TRUE;
		
	E_REQUEST_PROCESSING:
		DEBUG:='';
		FB_XML_PARSER.AppendAttributeAsInt(XML_HMIXML,'operationIndex',INDEX);
		FB_XML_PARSER.AppendAttributeAsInt(XML_HMIXML,'serviceId',2);		
		FB_XML_PARSER.SetChild(XML_ACTION,'2044',FALSE);
		XML_NODE := FB_XML_PARSER.AppendNode(XML_ARGUMENTS, 'SFC');
		FB_XML_PARSER.SetChild(XML_NODE,SFC,FALSE);
		
		FB_XML_PARSER.CopyDocument(REQUEST_STRING, SIZEOF(REQUEST_STRING));
		DEBUG:=REQUEST_STRING;
		STATE:= E_REQUEST_SEND;
		
	E_RESPONSE_PROCESSING:
		IF XML_REQUEST_RESULT.RESP_CODE = '0' THEN
			XML_RESTINFO:=FB_XML_PARSER.ChildByName(XML_RESULTS, 'RESTINFO');
			EXECUTE:=FALSE;
			STATE:= E_DISCONNECTING;
		ELSE
			MEMCPY(ADR(RESP),ADR(XML_REQUEST_RESULT), SIZEOF(XML_REQUEST_RESULT));
			ADSLOGSTR(ADSLOG_MSGTYPE_ERROR OR ADSLOG_MSGTYPE_LOG, 'SAP-ME error occured RESCODE: %s', CONCAT(CONCAT(RESP.RESP_CODE, ' ERR_MSG: '), RESP.ERR_MSG));
			EXECUTE:=FALSE;
			STATE:= E_DISCONNECTING;
		END_IF

END_CASE
SCRAP_SFC:= (STATE=E_DONE);
END_METHOD

METHOD PUBLIC SIGNOFF_SFC : BOOL
VAR_INPUT
	SFC:				STRING;
	INDEX:				INT;
END_VAR
VAR
	XML_NODE:				SXmlNode;
END_VAR
CASE STATE OF
	E_IDLE:
		EXECUTE:=TRUE;
		
	E_REQUEST_PROCESSING:
		FB_XML_PARSER.AppendAttributeAsInt(XML_HMIXML,'operationIndex',INDEX);
		FB_XML_PARSER.AppendAttributeAsInt(XML_HMIXML,'serviceId',2);	
		FB_XML_PARSER.SetChild(XML_ACTION,'3007',FALSE);
		XML_NODE := FB_XML_PARSER.AppendNode(XML_ARGUMENTS, 'SFC');
		FB_XML_PARSER.SetChild(XML_NODE,SFC,FALSE);
		
		FB_XML_PARSER.CopyDocument(REQUEST_STRING, SIZEOF(REQUEST_STRING));
		DEBUG:=REQUEST_STRING;
		STATE:= E_REQUEST_SEND;
		
	E_RESPONSE_PROCESSING:
		IF XML_REQUEST_RESULT.RESP_CODE = '0' THEN
			XML_RESTINFO:=FB_XML_PARSER.ChildByName(XML_RESULTS, 'RESTINFO');		
			EXECUTE:=FALSE;
			STATE:= E_DISCONNECTING;
		ELSE
			MEMCPY(ADR(RESP),ADR(XML_REQUEST_RESULT), SIZEOF(XML_REQUEST_RESULT));
			ADSLOGSTR(ADSLOG_MSGTYPE_ERROR OR ADSLOG_MSGTYPE_LOG, 'SAP-ME error occured RESCODE: %s', CONCAT(CONCAT(RESP.RESP_CODE, ' ERR_MSG: '), RESP.ERR_MSG));
			EXECUTE:=FALSE;
			STATE:= E_DISCONNECTING;
		END_IF
END_CASE
SIGNOFF_SFC:= (STATE=E_DONE);
END_METHOD

METHOD PUBLIC START_SFC : BOOL
VAR_INPUT
	SFC:				STRING;
	INDEX:				INT;
END_VAR
VAR
	XML_NODE:			SXmlNode;
END_VAR
CASE STATE OF
	E_IDLE:
		EXECUTE:=TRUE;
		
	E_REQUEST_PROCESSING:
		DEBUG:='';
		FB_XML_PARSER.AppendAttributeAsInt(XML_HMIXML,'operationIndex',INDEX);
		FB_XML_PARSER.AppendAttributeAsInt(XML_HMIXML,'serviceId',2);		
		FB_XML_PARSER.SetChild(XML_ACTION,'3010',FALSE);
		XML_NODE := FB_XML_PARSER.AppendNode(XML_ARGUMENTS, 'SFC');
		FB_XML_PARSER.SetChild(XML_NODE,SFC,FALSE);
		
		FB_XML_PARSER.CopyDocument(REQUEST_STRING, SIZEOF(REQUEST_STRING));
		DEBUG:=REQUEST_STRING;
		STATE:= E_REQUEST_SEND;
		
	E_RESPONSE_PROCESSING:
		IF XML_REQUEST_RESULT.RESP_CODE = '0' THEN
			XML_RESTINFO:=FB_XML_PARSER.ChildByName(XML_RESULTS, 'RESTINFO');
			EXECUTE:=FALSE;
			STATE:= E_DISCONNECTING;
		ELSE
			MEMCPY(ADR(RESP),ADR(XML_REQUEST_RESULT), SIZEOF(XML_REQUEST_RESULT));
			ADSLOGSTR(ADSLOG_MSGTYPE_ERROR OR ADSLOG_MSGTYPE_LOG, 'SAP-ME error occured RESCODE: %s', CONCAT(CONCAT(RESP.RESP_CODE, ' ERR_MSG: '), RESP.ERR_MSG));
			EXECUTE:=FALSE;
			STATE:= E_DISCONNECTING;
		END_IF

END_CASE
START_SFC:= (STATE=E_DONE);
END_METHOD

METHOD PUBLIC STOP_TIME_CONTROL : BOOL
VAR_INPUT
	SFCLIST:			STRING; //required Comma seperated list of SFCs ex.: "380027351822360103290549,380027351820360103290549"
	CONTROLTYPE:		STRING; //required Time Control Type Filter
	INDEX:				INT;
END_VAR
VAR
	XML_NODE:			SXmlNode;
END_VAR
CASE STATE OF
	E_IDLE:
		EXECUTE:=TRUE;
		
	E_REQUEST_PROCESSING:
		DEBUG:='';
		FB_XML_PARSER.AppendAttributeAsInt(XML_HMIXML,'operationIndex',INDEX);
		FB_XML_PARSER.AppendAttributeAsInt(XML_HMIXML,'serviceId',2);		
		FB_XML_PARSER.SetChild(XML_ACTION,'2014',FALSE);
		(* Set arguments *)
		XML_NODE := FB_XML_PARSER.AppendNode(XML_ARGUMENTS, 'SFCLIST');
		FB_XML_PARSER.SetChild(XML_NODE,SFCLIST,FALSE);
		XML_NODE := FB_XML_PARSER.AppendNode(XML_ARGUMENTS, 'CONTROLTYPE');
		FB_XML_PARSER.SetChild(XML_NODE,CONTROLTYPE,FALSE);
		
		FB_XML_PARSER.CopyDocument(REQUEST_STRING, SIZEOF(REQUEST_STRING));
		DEBUG:=REQUEST_STRING;
		STATE:= E_REQUEST_SEND;
		
	E_RESPONSE_PROCESSING:
		IF XML_REQUEST_RESULT.RESP_CODE = '0' THEN
			XML_RESTINFO:=FB_XML_PARSER.ChildByName(XML_RESULTS, 'RESTINFO');
			EXECUTE:=FALSE;
			STATE:= E_DISCONNECTING;
		ELSE
			MEMCPY(ADR(RESP),ADR(XML_REQUEST_RESULT), SIZEOF(XML_REQUEST_RESULT));
			ADSLOGSTR(ADSLOG_MSGTYPE_ERROR OR ADSLOG_MSGTYPE_LOG, 'SAP-ME error occured RESCODE: %s', CONCAT(CONCAT(RESP.RESP_CODE, ' ERR_MSG: '), RESP.ERR_MSG));
			EXECUTE:=FALSE;
			STATE:= E_DISCONNECTING;
		END_IF

END_CASE
STOP_TIME_CONTROL:= (STATE=E_DONE);
END_METHOD

METHOD PUBLIC VALIDATE_IN_BOM : BOOL
VAR_INPUT
	MATERIAL:				REFERENCE TO ST_MATERIAL;
	BOM:					REFERENCE TO ST_BOM;
	IS_VALID:				REFERENCE TO BOOL;
	RESULT_COMPONENT:		REFERENCE TO ST_BOM_COMPONENT;
END_VAR
VAR
	BOM_COMPONENT:			ST_BOM_COMPONENT;
	COMPONENT_MATERIAL:		ST_MATERIAL;
	CNT_BOM_COMPONENT:		INT;
	CNT_COMPONENT_MATERIAL:	INT;
	
	IS_VALID_REF:			BOOL;
END_VAR
IS_VALID_REF:=__ISVALIDREF(MATERIAL) AND __ISVALIDREF(BOM) AND __ISVALIDREF(IS_VALID) AND __ISVALIDREF(RESULT_COMPONENT);
IF IS_VALID_REF THEN
	IS_VALID:=FALSE;
	IF LEN(MATERIAL.MATERIAL)=11 AND LEN(MATERIAL.REVISION)=3 THEN
		FOR CNT_BOM_COMPONENT:=0 TO 19 BY 1 DO
			MEMCPY(ADR(BOM_COMPONENT),ADR(BOM.BOM_COMPONENTS[CNT_BOM_COMPONENT]), SIZEOF(BOM_COMPONENT));
			
			FOR CNT_COMPONENT_MATERIAL:=0 TO 9 BY 1 DO
				MEMCPY(ADR(COMPONENT_MATERIAL),ADR(BOM_COMPONENT.MATERIALS[CNT_COMPONENT_MATERIAL]), SIZEOF(COMPONENT_MATERIAL));
				
				IF COMPONENT_MATERIAL.MATERIAL=MATERIAL.MATERIAL AND COMPONENT_MATERIAL.REVISION= MATERIAL.REVISION THEN
					IS_VALID:=TRUE;
					MEMCPY(ADR(RESULT_COMPONENT),ADR(BOM_COMPONENT), SIZEOF(RESULT_COMPONENT));
					VALIDATE_IN_BOM:=TRUE;
				END_IF
			END_FOR;
		END_FOR;
		VALIDATE_IN_BOM:=TRUE;
	ELSE
		VALIDATE_IN_BOM:=TRUE;
	END_IF	
	RETURN;
ELSE
	VALIDATE_IN_BOM:=TRUE;
END_IF
END_METHOD

METHOD PRIVATE CREATE_XML_METH : BOOL
VAR_INPUT
END_VAR
FB_XML_PARSER.NewDocument();
OBJ_ROOT := FB_XML_PARSER.GetDocumentNode();
       
XML_HMIXML:= FB_XML_PARSER.AppendNode(OBJ_ROOT, 'HMI-XML');

	XML_PACKET:= FB_XML_PARSER.AppendNode(XML_HMIXML, 'PACKET');
	
		XML_BASICS:= FB_XML_PARSER.AppendNode(XML_PACKET, 'BASICS');
	
			XML_ACTION:= FB_XML_PARSER.AppendNode(XML_BASICS, 'ACTION');
				FB_XML_PARSER.SetChild(XML_ACTION,'',FALSE);	
				
		XML_ARGUMENTS:= FB_XML_PARSER.AppendNode(XML_PACKET, 'ARGUMENTS');	
			FB_XML_PARSER.SetChild(XML_ARGUMENTS,'',FALSE);
						
		XML_RESULTS:= FB_XML_PARSER.AppendNode(XML_PACKET, 'RESULTS');
			FB_XML_PARSER.SetChild(XML_RESULTS,'',FALSE);	
					
		XML_MSG:= FB_XML_PARSER.AppendNode(XML_PACKET, 'MSG');
			FB_XML_PARSER.SetChild(XML_MSG,'',FALSE);
END_METHOD

METHOD PUBLIC GET_LOCAL_TIME : STRING
VAR
	SYS_TIME:					DATE_AND_TIME;
	SYS_TIME_STRING	:			STRING;
	YEAR_STRING:				STRING[4];
	MONTH_STRING:				STRING[2];
	DAY_STRING:					STRING[2];
	TIME_STRING:				STRING;
	TIME_STAMP_STRING:			STRING;
	HOUR_STRING:				STRING;
END_VAR
GET_LOCAL_TIME:='';
SYS_TIME := SYSTEMTIME_TO_DT(TIMESTR:= SYS_TIME_FB.systemTime);
DAY_STRING:=MID((SYSTEMTIME_TO_STRING(SYS_TIME_FB.systemTime)),2,9);
MONTH_STRING:=MID((SYSTEMTIME_TO_STRING(SYS_TIME_FB.systemTime)),2,6);
YEAR_STRING:=MID((SYSTEMTIME_TO_STRING(SYS_TIME_FB.systemTime)),4,1);

IF SYS_TIME_FB.systemTime.wHour<10 THEN
	TIME_STRING:=MID((SYSTEMTIME_TO_STRING(SYS_TIME_FB.systemTime)),5,15);		
ELSE
	TIME_STRING:=MID((SYSTEMTIME_TO_STRING(SYS_TIME_FB.systemTime)),5,15);		
END_IF;	

IF SYS_TIME_FB.systemTime.wHour<13 THEN
	IF SYS_TIME_FB.systemTime.wHour=0 THEN
		HOUR_STRING:='12:';
	ELSE
		HOUR_STRING:=CONCAT(WORD_TO_STRING(SYS_TIME_FB.systemTime.wHour),':');
	END_IF	
	TIME_STRING:=CONCAT(TIME_STRING,' AM');
ELSE
	HOUR_STRING:=CONCAT(WORD_TO_STRING(SYS_TIME_FB.systemTime.wHour-12),':');
	TIME_STRING:=CONCAT(TIME_STRING,' PM');
END_IF	

TIME_STRING:=CONCAT(HOUR_STRING,TIME_STRING);	
TIME_STAMP_STRING:=CONCAT(CONCAT(CONCAT(MONTH_STRING,'/'),CONCAT(DAY_STRING,'/')),CONCAT(CONCAT(YEAR_STRING,' '),TIME_STRING));
	
GET_LOCAL_TIME:=TIME_STAMP_STRING;
RETURN;
END_METHOD

METHOD PRIVATE READ_XML_METH : BOOL
VAR_INPUT
END_VAR
IF RESPONSE_STRING<>'ERROR' THEN
OBJ_ROOT:= FB_XML_PARSER.ParseDocument(RESPONSE_STRING);
XML_HMIXML := FB_XML_PARSER.ChildByName(OBJ_ROOT, 'HMI-XML');
	XML_PACKET := FB_XML_PARSER.ChildByName(XML_HMIXML, 'PACKET');
		XML_BASICS := FB_XML_PARSER.ChildByName(XML_PACKET, 'BASICS');		
			XML_ACTION := FB_XML_PARSER.ChildByName(XML_BASICS, 'ACTION');
			FB_XML_PARSER.CopyNodeText(XML_ACTION, XML_REQUEST_RESULT.RESP_ACTION, SIZEOF(XML_REQUEST_RESULT.RESP_ACTION));				
		XML_ARGUMENTS := FB_XML_PARSER.ChildByName(XML_PACKET, 'ARGUMENTS');		
		XML_RESULTS := FB_XML_PARSER.ChildByName(XML_PACKET, 'RESULTS');			
		XML_MSG := FB_XML_PARSER.ChildByName(XML_PACKET, 'MSG');		
			XML_RESCODE := FB_XML_PARSER.ChildByName(XML_MSG, 'RESCODE');
			FB_XML_PARSER.CopyNodeText(XML_RESCODE, XML_REQUEST_RESULT.RESP_CODE, SIZEOF(XML_REQUEST_RESULT.RESP_CODE));				
			XML_RESSTANDARDMESSAGE := FB_XML_PARSER.ChildByName(XML_MSG, 'RESSTANDARDMESSAGE');
			FB_XML_PARSER.CopyNodeText(XML_RESSTANDARDMESSAGE, XML_REQUEST_RESULT.ERR_MSG, SIZEOF(XML_REQUEST_RESULT.ERR_MSG));
ELSE
	XML_REQUEST_RESULT.RESP_CODE:='-1';
	XML_REQUEST_RESULT.ERR_MSG:='Tcp communication error occured';
	XML_REQUEST_RESULT.RESP_ACTION:='-1';
END_IF
END_METHOD

ACTION FB_CALL_ACT:
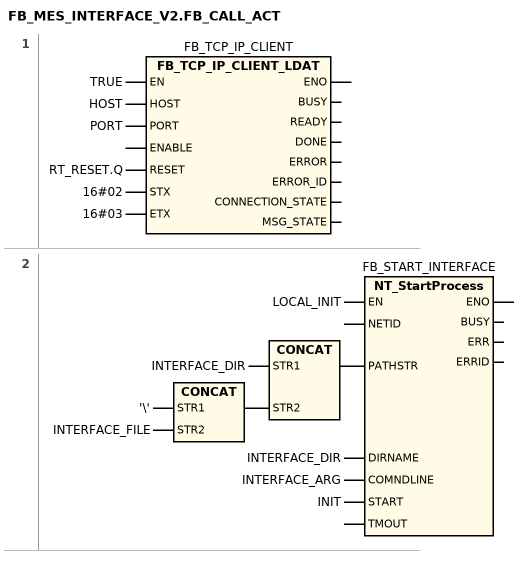
// NETWORK 1
FB_TCP_IP_CLIENT(HOST := HOST, PORT := PORT, RESET := RT_RESET.Q, STX := 16#02, ETX := 16#03); // FB_TCP_IP_CLIENT_LDAT

// NETWORK 2
IF LOCAL_INIT THEN
    FB_START_INTERFACE(
        PATHSTR := CONCAT(STR1 := INTERFACE_DIR, STR2 := CONCAT(STR1 := '\', STR2 := INTERFACE_FILE)),
        DIRNAME := INTERFACE_DIR,
        COMNDLINE := INTERFACE_ARG,
        START := INIT); // NT_StartProcess
END_IF
END_ACTION

END_FUNCTION_BLOCK

// FCs/FC_REMOVE_HEADER
FUNCTION FC_REMOVE_HEADER : STRING
VAR_INPUT
	INPUT:		STRING(255);
END_VAR
VAR
	HEADER_LENGTH:	INT;
END_VAR

FC_REMOVE_HEADER:=DELETE(INPUT, FIND(INPUT, ','), 1);

END_FUNCTION

// FCs/FC_GET_MATERIAL_FROM_HANDLE
FUNCTION FC_GET_MATERIAL_FROM_HANDLE : STRING
VAR_INPUT
	INPUT:			STRING;
END_VAR
VAR
END_VAR

FC_GET_MATERIAL_FROM_HANDLE:=LEFT(INPUT, 11);

END_FUNCTION

// FCs/FC_GET_REVISION_FROM_HANDLE
FUNCTION FC_GET_REVISION_FROM_HANDLE : STRING
VAR_INPUT
	INPUT:			STRING;
END_VAR
VAR
END_VAR

FC_GET_REVISION_FROM_HANDLE:=RIGHT(INPUT, 3);

END_FUNCTION

// FCs/FC_REMOVE_STRING
FUNCTION FC_REMOVE_STRING : STRING
VAR_INPUT
	VALUE:			STRING;			//Find this in source string 
	SOURCE:			STRING;			//Source string
END_VAR
VAR
	POSITION_OF_VALUE:		INT;	
	LENGTH_OF_VALUE:		INT;
END_VAR

POSITION_OF_VALUE:=FIND(SOURCE, VALUE);
LENGTH_OF_VALUE:=LEN(VALUE);
IF POSITION_OF_VALUE=0 OR LENGTH_OF_VALUE=0 THEN
	FC_REMOVE_STRING:=SOURCE;
	RETURN;
ELSE
	FC_REMOVE_STRING:=DELETE(SOURCE, LENGTH_OF_VALUE, POSITION_OF_VALUE);
END_IF

END_FUNCTION

// TESTs/GENERATE_MESDAT
FUNCTION GENERATE_MESDAT : BOOL
VAR_INPUT
	N:			INT:=1;
	MES:		REFERENCE TO FB_MES_INTERFACE_V2;
	MESDAT:		REFERENCE TO ST_MESDAT;
END_VAR
VAR
	CNT:		INT:=1;
	VAL:		LREAL;
	L_LIMIT:	LREAL;
	U_LIMIT:	LREAL;
	RAND:		DRAND;
END_VAR

MESDAT.N:=N;

FOR CNT:=1 TO N DO
	RAND(Seed:=0, Num=>VAL);
	VAL:=VAL*10;
	L_LIMIT:=(VAL-(VAL*0.1));
	U_LIMIT:=(VAL+(VAL*0.1));
	
    MESDAT.MESDAT[CNT].CLIENT_DATE:= MES.GET_LOCAL_TIME();
	MESDAT.MESDAT[CNT].VALUE:= LREAL_TO_FMTSTR(VAL, 4, TRUE);
	MESDAT.MESDAT[CNT].LL:= LREAL_TO_FMTSTR(L_LIMIT, 4, TRUE);
	MESDAT.MESDAT[CNT].UL:= LREAL_TO_FMTSTR(U_LIMIT, 4, TRUE);
	MESDAT.MESDAT[CNT].TEST_STATE:= '0';
	MESDAT.MESDAT[CNT].TEST_STEP:= INT_TO_STRING(CNT);
	MESDAT.MESDAT[CNT].UNIT:= 'UNIT';
	MESDAT.MESDAT[CNT].DESCR:= CONCAT('Test data DESC #', INT_TO_STRING(CNT));
END_FOR;

END_FUNCTION

// TESTs/GENERATE_NCDAT
FUNCTION GENERATE_NCDAT : BOOL;
VAR_INPUT
	N:			INT:=1;
	MES:		REFERENCE TO FB_MES_INTERFACE_V2;
	NCDAT:		REFERENCE TO ST_MESDAT;
END_VAR
VAR
	CNT:		INT:=1;
	VAL:		LREAL;
	L_LIMIT:	LREAL;
	U_LIMIT:	LREAL;
	RAND:		DRAND;
END_VAR

NCDAT.N:=N;

FOR CNT:=1 TO N DO
	RAND(Seed:=0, Num=>VAL);
	VAL:=VAL*10;
	L_LIMIT:=(VAL-(VAL*0.1));
	U_LIMIT:=(VAL+(VAL*0.1));
	
    NCDAT.MESDAT[CNT].CLIENT_DATE:= MES.GET_LOCAL_TIME();
	NCDAT.MESDAT[CNT].VALUE:= LREAL_TO_FMTSTR(VAL, 4, TRUE);
	NCDAT.MESDAT[CNT].LL:= LREAL_TO_FMTSTR(L_LIMIT, 4, TRUE);
	NCDAT.MESDAT[CNT].UL:= LREAL_TO_FMTSTR(U_LIMIT, 4, TRUE);
	NCDAT.MESDAT[CNT].RESPONSE_DESCRIPTION:= CONCAT('Test data DESC #', INT_TO_STRING(CNT));
	NCDAT.MESDAT[CNT].RESPONSE_CODE:= INT_TO_STRING(CNT*10);
	NCDAT.MESDAT[CNT].TEST_STATE:= '1';
	NCDAT.MESDAT[CNT].TEST_STEP:= INT_TO_STRING(CNT);
	NCDAT.MESDAT[CNT].UNIT:= 'UNIT';
	NCDAT.MESDAT[CNT].DESCR:= CONCAT('Test data DESC #', INT_TO_STRING(CNT));
END_FOR;

END_FUNCTION

// TESTs/HCP3_TEST_POU
PROGRAM HCP3_TEST_POU
VAR
	MES:						FB_MES_INTERFACE_V2;		(* Instance of MES-Interface function block *)
	RESP:						ST_REQUEST;				(* Reference to MES-Interface function block response *)
	INIT:						BOOL:=TRUE;
	RESET:						BOOL;					
	START:						BOOL;					
	STATE:						UDINT;
	INDEX:						INT;					
	
	COVER_BARCODE:				STRING:='288000060010020103725571';					(* COVER barcode *)
	COVER_PARENT:				STRING;					(* MRT parent barcode *)
	COVER_STATE:				ST_GET_OP_STATE;		(* Container of SFC State data which releated to Cover barcode *)
	COVER_INVENTORY:			ST_INVENTORY;			(* Result inventory of the import *)
	COVER_VALID:				BOOL;					
	
	CARRIER_BARCODE:			STRING:='288000000005020103725189';					(* CARRIER barcode *)
	CARRIER_PARENT:				STRING;					(* MRT parent barcode *)
	CARRIER_STATE:				ST_GET_OP_STATE;		(* Container of SFC State data which releated to Carrier barcode *)
	CARRIER_INVENTORY:			ST_INVENTORY;			(* Result inventory of the import *)
	CARRIER_VALID:				BOOL;					
	
	PCBA_BARCODE:				STRING:='380027351706990103944077';					(* 4010 PCBA barcode *)
	PCBA_PARENT:				STRING;					(* MRT parent barcode *)
	PCBA_STATE:					ST_GET_OP_STATE;		(* Container of SFC State data which releated to PCBA barcode *)
	PCBA_INVENTORY:				ST_INVENTORY;			(* Inventory data of PCBA *)
	PCBA_VALID:					BOOL;					
	PCBA_BOM:					ST_BOM;					(* Container of BOM releated to PCBA barcode *)
	PCBA_RECIPE:				STRING;
	PCBA_INVENTORY_LIST:		ST_INVENTORY_LIST;		(* Need to be filld with Inventory ID before try to assemble it *)
	PCBA_ASSY_RESULT:			E_TEST_STATE;			(* Assembly result Passed/Failed *)
	PCBA_CHECK_RESULT:			E_TEST_STATE;			(* Assembly result Passed/Failed *)
	PCBA_MATERIAL:				ST_MATERIAL;			(* Contains the PCBA material *)
	PCBA_SHOPORDER_LIST:		ST_SHOPORDER_LIST;		(* List of suitable sohoporder for the PCBA material *)
	
	FAN_BARCODE:				STRING:='288000000004000104014579';					(* FAN barcode *)
	FAN_PARENT:					STRING;					(* Parent of the FAN, need to be a PCBA barcode, with matching with BOM material. *)
	FAN_STATE:					ST_GET_OP_STATE;		(* Container of SFC State data which releated to Fan barcode *)
	FAN_INVENTORY:				ST_INVENTORY;			(* Result inventory of the import *)
	FAN_VALID:					BOOL;					
	
	MRT_BARCODE:				STRING;					(* MRT barcode *)
	MRT_STATE:					ST_GET_OP_STATE;		(* Container of SFC State data which releated to MRT barcode *)
	MRT_INVENTORY_LIST:			ST_INVENTORY_LIST;		(* Need to be filld with Inventory ID before try to assemble it *)
	MRT_ASSY_RESULT:			E_TEST_STATE;			(* Assembly result Passed/Failed *)
	MRT_BOM:					ST_BOM;					(* Container of BOM releated to PCBA barcode *)
	MRT_MATERIAL:				ST_MATERIAL;			(* Contains the MRT material *)
	MRT_MATERIAL_INFO:			ST_MATERIAL_INFO;		(* Contains the MRT material *)
	MRT_SHOPORDER_LIST:			ST_SHOPORDER_LIST;		(* List of suitable sohoporder for the MRT material *)
	
	(* Process variables *)		
	FAN_INSERT_CHECK_RESULT:		E_TEST_STATE;
	FAN_INSERT_CHECK_RECIPE:		STRING;
	
	FAN_CONNECTION_CEHCK_RESULT:	E_TEST_STATE;
	FAN_CONNECTION_CEHCK_RECIPE:	STRING;
	
	GAP_FILLER_CHECK_RESULT:		E_TEST_STATE;
	GAP_FILLER_CHECK_RECIPE:		STRING;
	
	GAP_FILLER_RESULT:				E_TEST_STATE;
	GAP_FILLER_RECIPE:				STRING;
	
	SCREWING_RESULT:				E_TEST_STATE;
	SCREWING_RECIPE:				STRING;
	
	(* Reusable variables*)
	(* Temporary containers for MES.GET_SHOPORDER_BY_MAT() *)

	SHOPORDER:					ST_SHOPORDER;
	RELEASE_COUNT:				STRING;
	
	(* Temporary containers for MES.VALIDATE_IN_BOM() *)
	COMPONENT_MATERIAL:			ST_MATERIAL;
	BOM_COMPONENT:				ST_BOM_COMPONENT;
	
	(*  *)
	MESDAT:						ST_MESDAT;
	NCDAT:						ST_MESDAT;
	
	
	DEBUG:						STRING(255);
	EXIT_INTERFACE:				BOOL;
	SHOW_INTERFACE:				BOOL;
	HIDE_INTERFACE:				BOOL;
END_VAR

MRT_MATERIAL.MATERIAL:='00003981088'; 	//Preconfigured by the opreator
MRT_MATERIAL.REVISION:='990';			//Preconfigured by the operator
RELEASE_COUNT:='1';						//Preconfigured by the operator - Required quantity.
IF INIT THEN
	(* Restart the SAP-ME Interface.exe on PLC restart. Or triggered on strange communication error. *)
	IF MES.LOCAL_INIT_SERVICE() THEN
		INIT:=FALSE;
	END_IF
ELSE
	IF EXIT_INTERFACE THEN
		(* TCP Request for exiting. *)
		IF MES.EXIT_SERVICE() THEN
			EXIT_INTERFACE:=FALSE;
		END_IF
	END_IF
	IF SHOW_INTERFACE THEN
		IF MES.SHOW_SERVICE() THEN
			SHOW_INTERFACE:=FALSE;
		END_IF
	END_IF
	IF HIDE_INTERFACE THEN
		IF MES.HIDE_SERVICE() THEN
			HIDE_INTERFACE:=FALSE;
		END_IF
	END_IF
	CASE STATE OF
	(* ###############################################################		Initialize		###########################################################################	*)
		0:			(* Material setup based on the selected material *)
			IF MES.GET_SHOPORDER_BY_MAT(MRT_MATERIAL, RELEASE_COUNT, INDEX, MRT_SHOPORDER_LIST) THEN
				STATE:=10;
			END_IF
		10: 		(* Slect ove suitable Shoporder - In this case work always with the idx:=0 *)
			IF MES.GET_TOTAL_BOM_BY_SO(MRT_SHOPORDER_LIST.LIST[0].HANDLE, INDEX, MRT_BOM) THEN
				STATE:=100;
			END_IF
	(* ###############################################################		Wait for start	###########################################################################	*)
		100:		(* Wait the start trigger *)
			IF START THEN
				INDEX:=0;
				STATE:=1000;
				START:=FALSE;
			END_IF				
	(* ################################################################################################################################################################
	   #
	   #
	   #																	ST10-Manual insertion
	   #
	   #
	   ################################################################################################################################################################ *)
	(* ###############################################################		Cover	insert	###########################################################################	*)
		1000:		(* Get current operation state of the cover *)
			IF MES.GET_CURRENT_OPERATION_STATE(COVER_BARCODE, INDEX, COVER_STATE) THEN 
				IF RESP.RESP_CODE='0' THEN
					IF COVER_STATE.OP_NAME='OP_GAP_FILLER_COVER' AND COVER_STATE.SFC_STATE='IN_QUEUE' AND COVER_STATE.OPEN_NC='FALSE' THEN
						COMPONENT_MATERIAL.MATERIAL:=COVER_STATE.MAT_NO;
						COMPONENT_MATERIAL.REVISION:=COVER_STATE.REVISION;
						
						COVER_INVENTORY.SFC:=COVER_BARCODE;
						COVER_INVENTORY.MAT_NO:=COVER_STATE.MAT_NO;
						COVER_INVENTORY.REVISION:=COVER_STATE.REVISION;
						
						STATE:=1030;
					ELSIF COVER_STATE.OP_NAME='NONE' AND COVER_STATE.SFC_STATE='UNKNOWN' AND COVER_STATE.OPEN_NC='FALSE' THEN
						STATE:=1010;
					ELSE
						DEBUG:='1000 - GET_OP_STATE() failed with wrong SFC_STATE or OPERATION';
						STATE:=99999;
					END_IF
				ELSE
					DEBUG:='1000 - GET_OP_STATE() failed with wrong rescode';
					STATE:=99999;
				END_IF
			END_IF
		1010:		(* Ipmort and pleace in_queue at the net operation OP_GAP_FILLER_COVER in my case is index[1].  *)
			INDEX:=1;
			IF MES.IMPORT_SFC(COVER_BARCODE, INDEX, COVER_INVENTORY) THEN
				IF RESP.RESP_CODE='0' THEN
					STATE:=1020;
				ELSE
					DEBUG:='1010 - ASSY_COMPLETE_SFC() failed with wrong rescode';
					STATE:=99999;
				END_IF
			END_IF
		1020:		(* Complet importing *)
			IF MES.COMPLETE_SFC(COVER_BARCODE, INDEX, E_TEST_STATE.PASSED) THEN
				IF RESP.RESP_CODE='0' THEN
					COMPONENT_MATERIAL.MATERIAL:=COVER_INVENTORY.MAT_NO;
					COMPONENT_MATERIAL.REVISION:=COVER_INVENTORY.REVISION;
					STATE:=1030;
				ELSE
					DEBUG:='1020 - ASSY_COMPLETE_SFC() failed with wrong rescode';
					STATE:=99999;
				END_IF
			END_IF
		1030:		(* validate cover in MRT BOM *)
			IF MES.VALIDATE_IN_BOM(COMPONENT_MATERIAL, MRT_BOM, COVER_VALID, BOM_COMPONENT) THEN
				IF COVER_VALID THEN
					//Set the cover parent to 0
					MEMSET(ADR(COVER_PARENT), 0, SIZEOF(COVER_PARENT));
					STATE:=1040;
				ELSE
					DEBUG:='VALIDATE_IN_BOM() cover is not part of the selected BOM';
					STATE:=99999;
				END_IF
			END_IF
		1040:		(* always check the parent, if have throw error to the opreator. *)
			IF MES.GET_INVENTORY_PARENT(COVER_BARCODE, INDEX, COVER_PARENT) THEN
				IF RESP.RESP_CODE='0' OR RESP.RESP_CODE='587' THEN
					IF COVER_PARENT='NONE' THEN
						STATE:=2000;
					ELSE
						DEBUG:='1050 - GET_PARENT() This cover has parent';
						STATE:=99999;
					END_IF
				ELSE
					DEBUG:='1050 - ASSY_GET_INVENTORY_PARENT() failed with wrong rescode';
					STATE:=99999;
				END_IF
			END_IF
			
	(* ###############################################################		Carrier	insert	###########################################################################	*)
		2000:		(* Carrier sequence *)
			MEMSET(ADR(MRT_INVENTORY_LIST), 0, SIZEOF(MRT_INVENTORY_LIST)); (* Clear inventory list *)
			IF MES.GET_CURRENT_OPERATION_STATE(CARRIER_BARCODE, INDEX, CARRIER_STATE) THEN
				IF RESP.RESP_CODE='0' THEN
					IF CARRIER_STATE.OP_NAME='NONE' AND CARRIER_STATE.SFC_STATE='DONE' AND CARRIER_STATE.OPEN_NC='FALSE' THEN (* If done the carrier must have parent barcode *)
						COMPONENT_MATERIAL.MATERIAL:=COVER_STATE.MAT_NO;
						COMPONENT_MATERIAL.REVISION:=COVER_STATE.REVISION;
						STATE:=2020;
					ELSIF CARRIER_STATE.OP_NAME='NONE' AND CARRIER_STATE.SFC_STATE='UNKNOWN' AND CARRIER_STATE.OPEN_NC='FALSE' THEN (* If unknown need to be import this new carrier *)
						STATE:=2010;
					ELSE
						DEBUG:='2000 - GET_OP_STATE() failed with wrong SFC_STATE or OPERATION';
						STATE:=99999;
					END_IF
				ELSE
					DEBUG:='2000 - GET_OP_STATE() failed with wrong rescode';
					STATE:=99999;
				END_IF
			END_IF
			
		2010:
			INDEX:=0;
			IF MES.IS_VALID_INVENTORY_AND_IMPORT(CARRIER_BARCODE, INDEX, CARRIER_INVENTORY) THEN (* Import new carrier *)
				IF RESP.RESP_CODE='0' THEN
					IF CARRIER_INVENTORY.DONE = 'TRUE' THEN
						COMPONENT_MATERIAL.MATERIAL:=CARRIER_INVENTORY.MAT_NO;
						COMPONENT_MATERIAL.REVISION:=CARRIER_INVENTORY.REVISION;
						DEBUG:='2000 - IS_VALID_INVENTORY_AND_IMPORT() passed, product imported, and done';
						STATE:=2020;
					ELSE
						DEBUG:='2000 - IS_VALID_INVENTORY_AND_IMPORT() failed, because it is not done';
						STATE:=99999;
					END_IF
				ELSE
					DEBUG:='2000 - IS_VALID_INVENTORY_AND_IMPORT() failed with wrong rescode';
					STATE:=99999;
				END_IF
			END_IF
		2020:
			IF MES.GET_INVENTORY_PARENT(CARRIER_BARCODE, INDEX, CARRIER_PARENT) THEN (* Get the parent barcode *)
				IF RESP.RESP_CODE='0' OR RESP.RESP_CODE='587' THEN
					IF CARRIER_PARENT<>'NONE' AND LEN(CARRIER_PARENT)=16 THEN
						MRT_BARCODE:=CARRIER_PARENT;
						STATE:=2030;
					ELSE
						STATE:=2030;
					END_IF
				ELSE
					DEBUG:='2020 - ASSY_GET_INVENTORY_PARENT() failed with wrong rescode';
					STATE:=99999;
				END_IF
			END_IF
		2030:
			IF MES.VALIDATE_IN_BOM(COMPONENT_MATERIAL, MRT_BOM, CARRIER_VALID, BOM_COMPONENT) THEN
				IF CARRIER_VALID THEN
					MRT_INVENTORY_LIST.LIST[0].SFC:=CARRIER_BARCODE;
					MEMSET(ADR(PCBA_PARENT), 0, SIZEOF(PCBA_PARENT));
					STATE:=3000;
				ELSE
					DEBUG:='VALIDATE_IN_BOM() cover is not part of the selected BOM';
					STATE:=99999;
				END_IF
			END_IF
			
	(* #################################################################	PCBA insert + FAN assy	###################################################################	*)		
		3000:		(* PCBA sequence *)
			IF MES.GET_INVENTORY_PARENT(PCBA_BARCODE, INDEX, PCBA_PARENT) THEN (* Get the parent barcode *)
				IF RESP.RESP_CODE='0' OR RESP.RESP_CODE='587' THEN
					IF PCBA_PARENT='NONE' THEN
						STATE:=3010;
					ELSE
						DEBUG:='3000 - ASSY_GET_INVENTORY_PARENT() This PCBA has parent';
						STATE:=99999;
					END_IF
				ELSE
					DEBUG:='3000 - ASSY_GET_INVENTORY_PARENT() failed with wrong rescode';
					STATE:=99999;
				END_IF
			END_IF
		3010:
			IF MES.GET_CURRENT_OPERATION_STATE(PCBA_BARCODE, INDEX, PCBA_STATE) THEN
				IF RESP.RESP_CODE='0' THEN
					
					PCBA_MATERIAL.MATERIAL:=PCBA_STATE.MAT_NO;
					PCBA_MATERIAL.REVISION:=PCBA_STATE.REVISION;
					STATE:=3020;
				ELSE
					DEBUG:='3010 - GET_CURRENT_OPERATION_STATE() failed with wrong rescode';
					STATE:=99999;
				END_IF
			END_IF
		3020:
			IF MES.VALIDATE_IN_BOM(PCBA_MATERIAL, MRT_BOM, PCBA_VALID, BOM_COMPONENT) THEN
				IF PCBA_VALID THEN
					IF PCBA_STATE.OP_NAME='OP_ASSEMBLY_2' AND PCBA_STATE.SFC_STATE='IN_QUEUE' AND PCBA_STATE.OPEN_NC='FALSE' THEN (* FAN Need to be assemble *)
						//assy fan + read
						INDEX:= STRING_TO_INT(PCBA_STATE.OP_INDEX);
						STATE:=3030;
					ELSIF PCBA_STATE.OP_NAME='NONE' AND PCBA_STATE.SFC_STATE='DONE' AND PCBA_STATE.OPEN_NC='FALSE' THEN (* PCA is pre-assembled, need to check parent *)
						// read fan
						STATE:=10000;
					ELSE
						DEBUG:='3020 - GET_CURRENT_OPERATION_STATE() failed with wrong SFC_STATE or OPERATION';
						STATE:=99999;
					END_IF
				ELSE
					DEBUG:='3020 - VALIDATE_IN_BOM() PCBA is not part of the selected BOM';
					STATE:=99999;
				END_IF
			END_IF		
		3030:		(* run trough this if PCBA in in queue on OP_ASSEMBLY_2 *)
			IF MES.GET_CURRENT_OPERATION_STATE(FAN_BARCODE, INDEX, FAN_STATE) THEN
				IF RESP.RESP_CODE='0' THEN
					IF FAN_STATE.OP_NAME='NONE' AND FAN_STATE.SFC_STATE='UNKNOWN' AND FAN_STATE.OPEN_NC='FALSE' THEN (* new fan need to be import for BOM check*)
						STATE:=3040;
					ELSIF FAN_STATE.OP_NAME='NONE' AND FAN_STATE.SFC_STATE='DONE' AND FAN_STATE.OPEN_NC='FALSE' THEN (* reused fan check parent barcode *)
						COMPONENT_MATERIAL.MATERIAL:=FAN_STATE.MAT_NO;
						COMPONENT_MATERIAL.REVISION:=FAN_STATE.REVISION;
						MEMSET(ADR(FAN_PARENT), 0, SIZEOF(FAN_PARENT));
						STATE:=3050;
					ELSE
						DEBUG:='3030 - GET_CURRENT_OPERATION_STATE() failed with wrong SFC_STATE or OPERATION';
						STATE:=99999;
					END_IF
				ELSE
					DEBUG:='3030 - GET_CURRENT_OPERATION_STATE() failed with wrong rescode';
					STATE:=99999;
				END_IF
			END_IF
		3040:
			INDEX:=0;
			IF MES.IS_VALID_INVENTORY_AND_IMPORT(FAN_BARCODE, INDEX, FAN_INVENTORY) THEN
				IF RESP.RESP_CODE='0' THEN
					IF FAN_INVENTORY.DONE = 'TRUE' THEN
						COMPONENT_MATERIAL.MATERIAL:=FAN_INVENTORY.MAT_NO;
						COMPONENT_MATERIAL.REVISION:=FAN_INVENTORY.REVISION;
						STATE:=3050;
					ELSE
						DEBUG:='3040 - IS_VALID_INVENTORY_AND_IMPORT() failed, because it is not done';
						STATE:=99999;
					END_IF
				ELSE
					DEBUG:='3040 - IS_VALID_INVENTORY_AND_IMPORT() failed with wrong rescode';
					STATE:=99999;
				END_IF
			END_IF
		3050:
			IF MES.GET_INVENTORY_PARENT(FAN_BARCODE, INDEX, FAN_PARENT) THEN (* Get the parent barcode *)
				IF RESP.RESP_CODE='0' OR RESP.RESP_CODE='587' THEN
					IF FAN_PARENT='NONE' THEN
						STATE:=3060;
					ELSE
						DEBUG:='3050 - ASSY_GET_INVENTORY_PARENT() This FAN has parent';
						STATE:=99999;
					END_IF
				ELSE
					DEBUG:='3050 - ASSY_GET_INVENTORY_PARENT() failed with wrong rescode';
					STATE:=99999;
				END_IF
			END_IF
		3060:
			IF MES.GET_SHOPORDER_BY_MAT(PCBA_MATERIAL, '1', INDEX, PCBA_SHOPORDER_LIST) THEN
				STATE:=3070;
			END_IF
		3070: 		(* Slect ove suitable Shoporder - In this case work always with the idx:=0 *)
			IF MES.GET_TOTAL_BOM_BY_SO(PCBA_SHOPORDER_LIST.LIST[0].HANDLE, INDEX, PCBA_BOM) THEN
				STATE:=3080;
			END_IF
		3080:
			IF MES.VALIDATE_IN_BOM(COMPONENT_MATERIAL, PCBA_BOM, FAN_VALID, BOM_COMPONENT) THEN
				IF FAN_VALID THEN
					MEMSET(ADR(PCBA_INVENTORY_LIST), 0, SIZEOF(PCBA_INVENTORY_LIST));
					STATE:=3090;
				ELSE
					DEBUG:='3080 - VALIDATE_IN_BOM() PCBA is not part of the selected BOM';
					STATE:=99999;
				END_IF
			END_IF
		3090:
			INDEX:=STRING_TO_INT(PCBA_STATE.OP_INDEX);
			PCBA_INVENTORY_LIST.LIST[0].MAT_NO:=COMPONENT_MATERIAL.MATERIAL;
			PCBA_INVENTORY_LIST.LIST[0].REVISION:=COMPONENT_MATERIAL.REVISION;
			PCBA_INVENTORY_LIST.LIST[0].SFC:=FAN_BARCODE;
			
			IF MES.START_SFC(PCBA_BARCODE, INDEX) THEN
				IF RESP.RESP_CODE='0' THEN
					STATE:=3095;
				ELSE
					DEBUG:='3090 - ASSY_START_SFC() failed with wrong rescode';
					STATE:=99999;
				END_IF
			END_IF
			
		3095: (* get recipe *)
			IF MES.GET_RECIPE_NAME_BY_OPERATION_XML('OP_ASSEMBLY_2', PCBA_RECIPE) THEN
				IF PCBA_RECIPE<>'' THEN
					//check fan
					STATE:=3100;
				ELSE
					DEBUG:='3090 - ASSY_START_SFC() failed with wrong rescode or empty recipe';
					STATE:=99999;
				END_IF
			END_IF
		3100:
			(* Assemble part (Fan into PCBA) *)
			IF MES.ASSEMBLE_BY_INVENTORY_LIST(PCBA_BARCODE, INDEX, PCBA_INVENTORY_LIST) THEN
				IF RESP.RESP_CODE='0' THEN
					PCBA_ASSY_RESULT:=E_TEST_STATE.PASSED;
				ELSE
					PCBA_ASSY_RESULT:=E_TEST_STATE.FAILED;
				END_IF
				STATE:=3110;
			END_IF
		3110:
			INDEX:=STRING_TO_INT(PCBA_STATE.OP_INDEX);
			IF MES.COMPLETE_SFC(PCBA_BARCODE, INDEX, PCBA_ASSY_RESULT) THEN
				IF RESP.RESP_CODE='0' THEN
					PCBA_INVENTORY.DONE:='FALSE';
					PCBA_INVENTORY.MAT_NO:=PCBA_MATERIAL.MATERIAL;
					PCBA_INVENTORY.REVISION:=PCBA_MATERIAL.REVISION;
					PCBA_INVENTORY.SFC:=PCBA_BARCODE;
					STATE:=10000;
				ELSE
					DEBUG:='3110 - ASSY_COMPLETE_SFC() failed with wrong rescode';
					STATE:=99999;
				END_IF
			END_IF		
		3120:
			IF MES.GET_INVENTORY_PARENT(FAN_BARCODE, INDEX, FAN_PARENT) THEN (* Get the parent barcode *)
				IF RESP.RESP_CODE='0' OR RESP.RESP_CODE='587' THEN
					IF FAN_PARENT=PCBA_BARCODE THEN
						STATE:=3200;
					ELSE
						DEBUG:='3120 - ASSY_GET_INVENTORY_PARENT() This FAN has parent';
						STATE:=99999;
					END_IF
				ELSE
					DEBUG:='3120 - ASSY_GET_INVENTORY_PARENT() failed with wrong rescode';
					STATE:=99999;
				END_IF
			END_IF		
	(* #################################################################	PCBA FAN assy check	###################################################################	*)			
		3200:		(* Start OP_AOI_PCBA_1 in my case is index[11]. *)
			INDEX:=11; // prepare the next operation
			IF MES.START_SFC(PCBA_BARCODE, INDEX) THEN
				IF RESP.RESP_CODE='0' THEN
					STATE:=3210;
				ELSE
					DEBUG:='3200 - ASSY_START_SFC() failed with wrong rescode';
					STATE:=99999;
				END_IF
			END_IF
		3210:
			IF MES.GET_RECIPE_NAME_BY_OPERATION_XML('OP_AOI_PCBA_2', FAN_INSERT_CHECK_RECIPE) THEN
				IF FAN_INSERT_CHECK_RECIPE<>'' THEN
					STATE:=3220;
				ELSE
					DEBUG:='3210 - ASSY_GET_RECIPE_NAME_BY_OPERATION() failed with wrong rescode or empty recipe';
					STATE:=99999;
				END_IF
			END_IF
		3220: 		(* set result of FAN connection check *)	
			FAN_INSERT_CHECK_RESULT:=E_TEST_STATE.PASSED;
			STATE:=3230;		
		3230:		(* Complete OP_AOI_PCBA_1 in my case is index[11]. *)
			IF MES.COMPLETE_SFC(PCBA_BARCODE, INDEX, FAN_INSERT_CHECK_RESULT) THEN
				IF RESP.RESP_CODE='0' THEN
					STATE:=10000;
				ELSE
					DEBUG:='3230 - ASSY_COMPLETE_SFC() failed with wrong rescode';
					STATE:=99999;
				END_IF
			END_IF	
		
	(* ################################################################################################################################################################
	   #
	   #
	   #																	ST11-Labeling
	   #
	   #
	   ################################################################################################################################################################ *)
	(* ##############################################################		Generate MRT and print label	###########################################################	*)
		10000: 
			IF MRT_BARCODE='' THEN
				STATE:=10010;
			ELSE
				STATE:=10070;
			END_IF
			
		10010: 		(* Generate new MRT barcode if not exist yet - This call need to be call at OP_GET_MRT operation in my case is index[13]. *)
			INDEX:=13; // prepare the next operation
			IF MES.GENERATE_SFC_BY_SO_AND_START(MRT_MATERIAL_INFO, 'TRUE', 'TRUE', MRT_BARCODE, INDEX) THEN
				IF RESP.RESP_CODE='0' THEN
					INDEX:=12; // prepare the next operation
					STATE:=10020;
				ELSE
					DEBUG:='10010 - ASSY_COMPLETE_SFC() failed with wrong rescode';
					STATE:=99999;
				END_IF
			END_IF
			
		10020:		(* Start OP_GET_MRT_LABEL in my case is index[12]. *)
			IF MES.START_SFC(MRT_BARCODE, INDEX) THEN
				IF RESP.RESP_CODE='0' THEN
					STATE:=10030;
				ELSE
					DEBUG:='10020 - ASSY_START_SFC() failed with wrong rescode';
					STATE:=99999;
				END_IF
			END_IF
			
		10030:		(* Complete OP_GET_MRT_LABEL in my case is index[12]. *)
			IF MES.COMPLETE_SFC(MRT_BARCODE, INDEX, E_TEST_STATE.PASSED) THEN
				IF RESP.RESP_CODE='0' THEN
					STATE:=10040;
				ELSE
					DEBUG:='10030 - ASSY_COMPLETE_SFC() failed with wrong rescode';
					STATE:=99999;
				END_IF
			END_IF
			
	(* ##############################################################		Assemble carrier into MRT	###############################################################	*)		
		10040:		(* Start OP_ASSY_AUTO_1 in my case is index[6]. *)
			INDEX:=6; // prepare the next operation
			IF MES.START_SFC(MRT_BARCODE, INDEX) THEN
				IF RESP.RESP_CODE='0' THEN
					STATE:=10050;
				ELSE
					DEBUG:='10040 - ASSY_START_SFC() failed with wrong rescode';
					STATE:=99999;
				END_IF
			END_IF
			
		10050: 		(* Assemble part (Carrier into MRT) *)
			MRT_ASSY_RESULT:=E_TEST_STATE.FAILED;
			IF MES.ASSEMBLE_BY_INVENTORY_LIST(MRT_BARCODE, INDEX, MRT_INVENTORY_LIST) THEN
				IF RESP.RESP_CODE='0' THEN
					MRT_ASSY_RESULT:=E_TEST_STATE.PASSED;
				ELSE
					MRT_ASSY_RESULT:=E_TEST_STATE.FAILED;
				END_IF
				STATE:=10060;
			END_IF	
			
		10060:		(* Complete OP_ASSY_AUTO_1 in my case is index[6]. *)
			IF MES.COMPLETE_SFC(MRT_BARCODE, INDEX, MRT_ASSY_RESULT) THEN
				IF RESP.RESP_CODE='0' THEN
					STATE:=10070;
					MRT_INVENTORY_LIST.LIST[0]:=PCBA_INVENTORY;
					MRT_INVENTORY_LIST.LIST[1]:=COVER_INVENTORY;
				ELSE
					DEBUG:='10060 - ASSY_COMPLETE_SFC() failed with wrong rescode';
					STATE:=99999;
				END_IF
			END_IF
			
	(* ##############################################################		FAN connection check	###################################################################	*)		
		10070:		(* Start OP_AOI_PCBA_2 in my case is index[14]. *)
			INDEX:=11; // prepare the next operation
			IF MES.START_SFC(PCBA_BARCODE, INDEX) THEN
				IF RESP.RESP_CODE='0' THEN
					STATE:=10080;
				ELSE
					DEBUG:='10040 - ASSY_START_SFC() failed with wrong rescode';
					STATE:=99999;
				END_IF
			END_IF
		10080:
			IF MES.GET_RECIPE_NAME_BY_OPERATION_XML('OP_AOI_PCBA_2', FAN_CONNECTION_CEHCK_RECIPE) THEN
				IF FAN_CONNECTION_CEHCK_RECIPE<>'' THEN
					STATE:=20020;
				ELSE
					DEBUG:='20010 - ASSY_GET_RECIPE_NAME_BY_OPERATION() failed with wrong rescode or empty recipe';
					STATE:=99999;
				END_IF
			END_IF
		10090: 		(* set result of FAN connection check *)	
			FAN_CONNECTION_CEHCK_RESULT:=E_TEST_STATE.PASSED;
			STATE:=10100;		
		10100:		(* Complete OP_AOI_PCBA_2 in my case is index[14]. *)
			IF MES.COMPLETE_SFC(PCBA_BARCODE, INDEX, FAN_CONNECTION_CEHCK_RESULT) THEN
				IF RESP.RESP_CODE='0' THEN
					STATE:=10070;
					MRT_INVENTORY_LIST.LIST[0]:=PCBA_INVENTORY;
				ELSE
					DEBUG:='10060 - ASSY_COMPLETE_SFC() failed with wrong rescode';
					STATE:=99999;
				END_IF
			END_IF
	(* ################################################################################################################################################################
	   #
	   #
	   #																	ST20-Gapfiller
	   #
	   #
	   ################################################################################################################################################################ *)
	(* ##############################################################		Cover dispensing 		###################################################################	*)
		20000:		(* Start OP_GAP_FILLER_COVER in my case is index[1]. *)
			GAP_FILLER_RESULT:=E_TEST_STATE.FAILED;
			INDEX:=1; // prepare the next operation
			IF MES.START_SFC(COVER_BARCODE, INDEX) THEN
				IF RESP.RESP_CODE='0' THEN
					STATE:=20010;
				ELSE
					DEBUG:='20000 - ASSY_START_SFC() failed with wrong rescode';
					STATE:=99999;
				END_IF
			END_IF
		20010: 		(* Get ricpe name *)
			IF MES.GET_RECIPE_NAME_BY_OPERATION_XML('OP_GAP_FILLER_COVER', GAP_FILLER_RECIPE) THEN
				IF GAP_FILLER_RECIPE<>'' THEN
					STATE:=20020;
				ELSE
					DEBUG:='20010 - ASSY_GET_RECIPE_NAME_BY_OPERATION() failed with wrong rescode or empty recipe';
					STATE:=99999;
				END_IF
			END_IF
			
		20020: 		(* Dispensing the material...then set result. *)
			(* !Important - Do not execute the remaining dispensing if failed.  *)
			GAP_FILLER_RESULT:=E_TEST_STATE.PASSED;
			STATE:=20030;	
			
		20030:		(* Complete OP_GAP_FILLER_COVER in my case is index[2]. *)
			IF MES.COMPLETE_SFC(COVER_BARCODE, INDEX, GAP_FILLER_RESULT) THEN
				IF RESP.RESP_CODE='0' THEN
					(* Result passed then *)
					MRT_INVENTORY_LIST.LIST[1]:=COVER_INVENTORY;
					STATE:=20100;
				ELSE
					DEBUG:='20030 - ASSY_COMPLETE_SFC() failed with wrong rescode';
					STATE:=99999;
				END_IF
			END_IF
	(* ##############################################################		MRT 1 dispensing 		###################################################################	*)
		20100:		(* Start OP_GAP_FILLER_MRT_1 in my case is index[2]. *)
			INDEX:=2; // prepare the next operation
			IF MES.START_SFC(MRT_BARCODE, INDEX) THEN
				IF RESP.RESP_CODE='0' THEN
					STATE:=20010;
				ELSE
					DEBUG:='20000 - ASSY_START_SFC() failed with wrong rescode';
					STATE:=99999;
				END_IF
			END_IF
		20110: 		(* Get ricpe name *)
			IF MES.GET_RECIPE_NAME_BY_OPERATION_XML('OP_GAP_FILLER_MRT_1', GAP_FILLER_RECIPE) THEN
				IF GAP_FILLER_RECIPE<>'' THEN
					STATE:=20020;
				ELSE
					DEBUG:='20010 - ASSY_GET_RECIPE_NAME_BY_OPERATION() failed with wrong rescode or empty recipe';
					STATE:=99999;
				END_IF
			END_IF
			
		20120: 		(* Dispensing the material...then set result. *)
			(* !Important - Do not execute the remaining dispensing if failed.  *)
			GAP_FILLER_RESULT:=E_TEST_STATE.PASSED;
			STATE:=20030;	
			
		20130:		(* Complete OP_GAP_FILLER_MRT_1 in my case is index[2]. *)
			IF MES.COMPLETE_SFC(MRT_BARCODE, INDEX, GAP_FILLER_RESULT) THEN
				IF RESP.RESP_CODE='0' THEN
					STATE:=20200;
				ELSE
					DEBUG:='20130 - ASSY_COMPLETE_SFC() failed with wrong rescode';
					STATE:=99999;
				END_IF
			END_IF
	(* ##############################################################		MRT 2 dispensing 		###################################################################	*)
		20200:		(* Start OP_GAP_FILLER_MRT_2 in my case is index[3]. *)
			INDEX:=3; // prepare the next operation
			IF MES.START_SFC(MRT_BARCODE, INDEX) THEN
				IF RESP.RESP_CODE='0' THEN
					STATE:=20210;
				ELSE
					DEBUG:='20200 - ASSY_START_SFC() failed with wrong rescode';
					STATE:=99999;
				END_IF
			END_IF
		20210: 		(* Get ricpe name *)
			IF MES.GET_RECIPE_NAME_BY_OPERATION_XML('OP_GAP_FILLER_MRT_2', GAP_FILLER_RECIPE) THEN
				IF GAP_FILLER_RECIPE<>'' THEN
					STATE:=20220;
				ELSE
					DEBUG:='20210 - ASSY_GET_RECIPE_NAME_BY_OPERATION() failed with wrong rescode or empty recipe';
					STATE:=99999;
				END_IF
			END_IF
			
		20220: 		(* Dispensing the material...then set result. *)
			(* !Important - Do not execute the remaining dispensing if failed.  *)
			GAP_FILLER_RESULT:=E_TEST_STATE.PASSED;
			STATE:=20230;	
			
		20230:		(* Complete OP_GAP_FILLER_MRT_2 in my case is index[3]. *)
			IF MES.COMPLETE_SFC(MRT_BARCODE, INDEX, GAP_FILLER_RESULT) THEN
				IF RESP.RESP_CODE='0' THEN
					STATE:=30000;
				ELSE
					DEBUG:='20230 - ASSY_COMPLETE_SFC() failed with wrong rescode';
					STATE:=99999;
				END_IF
			END_IF
	(* ################################################################################################################################################################
	   #
	   #
	   #																	ST40-Automatic assembly
	   #
	   #
	   ################################################################################################################################################################ *)
	(* ##############################################################		MRT/Cover dispensing check 		###################################################################	*)
		30000:		(* Start OP_GAP_FILLER_CHECK in my case is index[4]. *)
			GAP_FILLER_CHECK_RESULT:=E_TEST_STATE.FAILED;
			INDEX:=4; // prepare the next operation
			IF MES.START_SFC(MRT_BARCODE, INDEX) THEN
				IF RESP.RESP_CODE='0' THEN
					STATE:=30010;
				ELSE
					DEBUG:='30000 - ASSY_START_SFC() failed with wrong rescode';
					STATE:=99999;
				END_IF
			END_IF
		30010: 		(* Get ricpe name *)
			IF MES.GET_RECIPE_NAME_BY_OPERATION_XML('OP_GAP_FILLER_CHECK', GAP_FILLER_CHECK_RECIPE) THEN
				IF GAP_FILLER_CHECK_RECIPE<>'' THEN
					STATE:=30020;
				ELSE
					DEBUG:='30010 - ASSY_GET_RECIPE_NAME_BY_OPERATION() failed with wrong rescode or empty recipe';
					STATE:=99999;
				END_IF
			END_IF
			
		30020: 		(* Check dispensing quality... then set result. *)
			GAP_FILLER_CHECK_RESULT:=E_TEST_STATE.PASSED;
			STATE:=30030;	
			
		30030:		(* Complete OP_GAP_FILLER_CHECK in my case is index[4]. *)
			IF MES.COMPLETE_SFC(MRT_BARCODE, INDEX, GAP_FILLER_CHECK_RESULT) THEN
				IF RESP.RESP_CODE='0' THEN
					MRT_INVENTORY_LIST.LIST[1]:=COVER_INVENTORY;
					STATE:=30200;
				ELSE
					DEBUG:='30030 - ASSY_COMPLETE_SFC() failed with wrong rescode';
					STATE:=99999;
				END_IF
			END_IF
	(* ##############################################################		MRT final assembly 		###################################################################	*)
		30200:		(* Start OP_ASSY_AUTO_2 in my case is index[7]. *)
			INDEX:=7; // prepare the next operation, the inventory list is filled currently.
			IF MES.START_SFC(MRT_BARCODE, INDEX) THEN
				IF RESP.RESP_CODE='0' THEN
					STATE:=30210;
				ELSE
					DEBUG:='30200 - ASSY_START_SFC() failed with wrong rescode';
					STATE:=99999;
				END_IF
			END_IF
			
		30210: 		(* Assemble parts (PCBA and Cover into MRT) *)
			IF MES.ASSEMBLE_BY_INVENTORY_LIST(MRT_BARCODE, INDEX, MRT_INVENTORY_LIST) THEN
				IF RESP.RESP_CODE='0' THEN
					STATE:=30210;
					MRT_ASSY_RESULT:=E_TEST_STATE.PASSED;
				ELSE
					STATE:=30220; // jump to scrap
					MRT_ASSY_RESULT:=E_TEST_STATE.FAILED;
				END_IF
				
			END_IF	
		30220:		(* Scrap the PCBA if needed *)	
			IF MES.SCRAP_SFC(PCBA_BARCODE, INDEX) THEN
				DEBUG:='30220 - PCBA is scraped';
				STATE:=99999;
			END_IF
			
		30230:		(* Complete OP_ASSY_AUTO_2 in my case is index[7]. *)
			IF MES.COMPLETE_SFC(MRT_BARCODE, INDEX, MRT_ASSY_RESULT) THEN
				IF RESP.RESP_CODE='0' THEN
					STATE:=40000;
				ELSE
					DEBUG:='30230 - ASSY_COMPLETE_SFC() failed with wrong rescode';
					STATE:=99999;
				END_IF
			END_IF
	(* ################################################################################################################################################################
	   #
	   #
	   #																	ST50-Screwing
	   #
	   #
	   ################################################################################################################################################################ *)
	(* ##############################################################			MRT 1 screwing 		###################################################################	*)
		40000:		(* Start OP_SCREWING_AUTO_1 in my case is index[9]. *)
		
			//Generate random MEASUREMENT data
			MEMSET(ADR(MESDAT), 0, SIZEOF(MESDAT));
			GENERATE_MESDAT(10, MES, MESDAT);
			
			//Generate random NC data
			MEMSET(ADR(NCDAT), 0, SIZEOF(NCDAT));
			GENERATE_NCDAT(1, MES, NCDAT);
			
			INDEX:=9; // prepare the next operation
			IF MES.START_SFC(MRT_BARCODE, INDEX) THEN
				IF RESP.RESP_CODE='0' THEN
					STATE:=40010;
				ELSE
					DEBUG:='20000 - ASSY_START_SFC() failed with wrong rescode';
					STATE:=99999;
				END_IF
			END_IF
		40010: 		(* Get ricpe name *)
			IF MES.GET_RECIPE_NAME_BY_OPERATION_XML('OP_SCREWING_AUTO_1', SCREWING_RECIPE) THEN
				IF SCREWING_RECIPE<>'' THEN
					STATE:=40020;
				ELSE
					DEBUG:='20010 - ASSY_GET_RECIPE_NAME_BY_OPERATION() failed with wrong rescode or empty recipe';
					STATE:=99999;
				END_IF
			END_IF
			
		40020: 	
			SCREWING_RESULT:=E_TEST_STATE.PASSED;
			IF SCREWING_RESULT=E_TEST_STATE.PASSED THEN
				STATE:=40030;
			ELSE
				STATE:=40040;
			END_IF	
		40030:		(* Log NonConformance data *)
			IF MES.ASSY_SAVE_NCDAT(MRT_BARCODE, INDEX, NCDAT) THEN
				IF RESP.RESP_CODE = '0' THEN
					STATE:=40040;
				ELSE
					DEBUG:='40030 - SAVE_NCDAT() failed with wrong rescode';
					STATE:=99999;
				END_IF
			END_IF
		40040:		(* Log Measurement data if failed *)
			IF MES.ASSY_SAVE_MESDAT(MRT_BARCODE, INDEX, MESDAT) THEN
				IF RESP.RESP_CODE = '0' THEN
					STATE:=40050;
				ELSE
					DEBUG:='40040 - SAVE_MESDAT() failed with wrong rescode';
					STATE:=99999;
				END_IF			
			END_IF	
		40050:		(* Complete OP_SCREWING_AUTO_1 in my case is index[9]. *)
			IF MES.COMPLETE_SFC(MRT_BARCODE, INDEX, SCREWING_RESULT) THEN
				IF RESP.RESP_CODE='0' THEN
					STATE:=40100;
				ELSE
					DEBUG:='40050 - ASSY_COMPLETE_SFC() failed with wrong rescode';
					STATE:=99999;
				END_IF
			END_IF
	(* ##############################################################			MRT 2 screwing 		###################################################################	*)
		40100:		(* Start OP_SCREWING_AUTO_2 in my case is index[10]. *)
		
				//Generate random MEASUREMENT data
			MEMSET(ADR(MESDAT), 0, SIZEOF(MESDAT));
			GENERATE_MESDAT(10, MES, MESDAT);
			
			//Generate random NC data
			MEMSET(ADR(NCDAT), 0, SIZEOF(NCDAT));
			GENERATE_NCDAT(1, MES, NCDAT);
			
			INDEX:=10; // prepare the next operation
			IF MES.START_SFC(MRT_BARCODE, INDEX) THEN
				IF RESP.RESP_CODE='0' THEN
					STATE:=40110;
				ELSE
					DEBUG:='40100 - ASSY_START_SFC() failed with wrong rescode';
					STATE:=99999;
				END_IF
			END_IF
		40110: 		(* Get ricpe name *)
			IF MES.GET_RECIPE_NAME_BY_OPERATION_XML('OP_SCREWING_AUTO_2', SCREWING_RECIPE) THEN
				IF GAP_FILLER_RECIPE<>'' THEN
					STATE:=40120;
				ELSE
					DEBUG:='40110 - ASSY_GET_RECIPE_NAME_BY_OPERATION() failed with wrong rescode or empty recipe';
					STATE:=99999;
				END_IF
			END_IF
			
